// TwinCAT 3 PLC project Untitled1
// ProgramVersion: 3.1.4023.0
// libraries:
//   Tc2_Math, * (Beckhoff Automation GmbH)
//   Tc2_Standard, * (Beckhoff Automation GmbH)
//   Tc2_System, * (Beckhoff Automation GmbH)
//   Tc3_Mc3PlanarMotion, * (Beckhoff Automation GmbH)
//   Tc3_Module, * (Beckhoff Automation GmbH)
//   Tc3_Physics, * (Beckhoff Automation GmbH)
//   XboxControllerUtilities, * (Beckhoff Community)
// project tree:
//   / PlcTask.TcTTO
//   POUs/ MAIN.TcPOU
// real-time tasks:
//   TASK XPlanar Task3: cycle T#250us, priority 1, ADS port 350
//   TASK XPlanar Task4: cycle T#250us, priority 2, ADS port 351
//   TASK Job Task: cycle default, priority 32
//   TASK MC-Task (MET): cycle T#250us, priority 6, ADS port 521
//   TASK MC-Task (MPT): cycle T#10ms, priority 8, ADS port 531
//   TASK PlcTask: cycle T#250us, priority 20, ADS port 352
// I/O:
//   DEVICE Device 1 (EtherCAT) (disabled), AmsNetId 169.254.25.219.2.1
//     Term 1 (EK1200) [EK1200-5000 EtherCAT Power supply (2A E-Bus)]
//       Term 2 (EL9222-9482) [EL9222-9482 Overcurrent protection 24V DC, 2Ch., 8A/2A]
//       Term 3 (EL9222-6600) [EL9222-6600 Overcurrent protection 24V DC, 2Ch., max. 4A, adjustable]
//       Term 4 (EL9011) [EL9011 End Terminal]
//   DEVICE Device 6 (EtherCAT), AmsNetId 169.254.25.219.7.1
//     Term 5 (APS4322-7000) [APS4322-7000 Drive]
//       Term 6 (APS4322-5000) [APS4322-5000 Feedback]
//     Term 7 (APS4322-7000) [APS4322-7000 Drive]
//       Term 8 (APS4322-5000) [APS4322-5000 Feedback]
//     Term 9 (APS4322-7000) [APS4322-7000 Drive]
//       Term 10 (APS4322-5000) [APS4322-5000 Feedback]
//     Term 11 (APS4322-7000) [APS4322-7000 Drive]
//       Term 12 (APS4322-5000) [APS4322-5000 Feedback]
//     Term 13 (APS4322-7000) [APS4322-7000 Drive]
//       Term 14 (APS4322-5000) [APS4322-5000 Feedback]
//     Term 15 (APS4322-7000) [APS4322-7000 Drive]
//       Term 16 (APS4322-5000) [APS4322-5000 Feedback]
//   DEVICE Device 2 (EtherCAT), AmsNetId 169.254.25.219.3.1
//     Term 17 (APS4322-7000) [APS4322-7000 Drive]
//       Term 18 (APS4322-5000) [APS4322-5000 Feedback]
//     Term 19 (APS4322-7000) [APS4322-7000 Drive]
//       Term 20 (APS4322-5000) [APS4322-5000 Feedback]
//     Term 21 (APS4322-7000) [APS4322-7000 Drive]
//       Term 22 (APS4322-5000) [APS4322-5000 Feedback]
//     Term 23 (APS4322-7000) [APS4322-7000 Drive]
//       Term 24 (APS4322-5000) [APS4322-5000 Feedback]
//     Term 25 (APS4322-7000) [APS4322-7000 Drive]
//       Term 26 (APS4322-5000) [APS4322-5000 Feedback]
//     Term 27 (APS4322-7000) [APS4322-7000 Drive]
//       Term 28 (APS4322-5000) [APS4322-5000 Feedback]
// variable links:
//   Device 2 (EtherCAT) <-> TcCOM Objects/XPlanar/Part1/Tile1
//     Term 17 (APS4322-7000)/APS Comm Inputs/CommStatusWord <-> Data Pointer/MoverCommStatusWord
//     Term 17 (APS4322-7000)/APS Comm Inputs/Data {1..4} <-> Data Pointer/MoverCommDataIn[{0..3}]  (4 links)
//     Term 17 (APS4322-7000)/APS Comm Outputs/CommControlWord <-> Data Pointer/MoverCommControlWord
//     Term 17 (APS4322-7000)/APS Comm Outputs/Data 1 <-> Data Pointer/MoverCommDataOut
//     Term 17 (APS4322-7000)/APS Diagdata/DC Link Voltage <-> Data Pointer/DcLinkVoltage
//     Term 17 (APS4322-7000)/APS Diagdata/Power supply current <-> Data Pointer/PowerSupplyCurrent
//     Term 17 (APS4322-7000)/APS Inputs/StatusWord <-> Data Pointer/PowerUnitStatusWord
//     Term 17 (APS4322-7000)/APS Outputs/ControlWord <-> Data Pointer/PowerUnitControlWord
//     Term 17 (APS4322-7000)/APS Outputs/Current D 0X0 <-> Data Pointer/DCurrentSetPoints[0]
//     Term 17 (APS4322-7000)/APS Outputs/Current D 0X1 <-> Data Pointer/DCurrentSetPoints[1]
//     Term 17 (APS4322-7000)/APS Outputs/Current D 0X2 <-> Data Pointer/DCurrentSetPoints[2]
//     Term 17 (APS4322-7000)/APS Outputs/Current D 1X0 <-> Data Pointer/DCurrentSetPoints[6]
//     Term 17 (APS4322-7000)/APS Outputs/Current D 1X1 <-> Data Pointer/DCurrentSetPoints[7]
//     Term 17 (APS4322-7000)/APS Outputs/Current D 1X2 <-> Data Pointer/DCurrentSetPoints[8]
//     Term 17 (APS4322-7000)/APS Outputs/Current D 2X0 <-> Data Pointer/DCurrentSetPoints[12]
//     Term 17 (APS4322-7000)/APS Outputs/Current D 2X1 <-> Data Pointer/DCurrentSetPoints[13]
//     Term 17 (APS4322-7000)/APS Outputs/Current D 2X2 <-> Data Pointer/DCurrentSetPoints[14]
//     Term 17 (APS4322-7000)/APS Outputs/Current D 3X0 <-> Data Pointer/DCurrentSetPoints[18]
//     Term 17 (APS4322-7000)/APS Outputs/Current D 3X1 <-> Data Pointer/DCurrentSetPoints[19]
//     Term 17 (APS4322-7000)/APS Outputs/Current D 3X2 <-> Data Pointer/DCurrentSetPoints[20]
//     Term 17 (APS4322-7000)/APS Outputs/Current D 0Y0 <-> Data Pointer/DCurrentSetPoints[3]
//     Term 17 (APS4322-7000)/APS Outputs/Current D 0Y1 <-> Data Pointer/DCurrentSetPoints[4]
//     Term 17 (APS4322-7000)/APS Outputs/Current D 0Y2 <-> Data Pointer/DCurrentSetPoints[5]
//     Term 17 (APS4322-7000)/APS Outputs/Current D 1Y0 <-> Data Pointer/DCurrentSetPoints[9]
//     Term 17 (APS4322-7000)/APS Outputs/Current D 1Y1 <-> Data Pointer/DCurrentSetPoints[10]
//     Term 17 (APS4322-7000)/APS Outputs/Current D 1Y2 <-> Data Pointer/DCurrentSetPoints[11]
//     Term 17 (APS4322-7000)/APS Outputs/Current D 2Y0 <-> Data Pointer/DCurrentSetPoints[15]
//     Term 17 (APS4322-7000)/APS Outputs/Current D 2Y1 <-> Data Pointer/DCurrentSetPoints[16]
//     Term 17 (APS4322-7000)/APS Outputs/Current D 2Y2 <-> Data Pointer/DCurrentSetPoints[17]
//     Term 17 (APS4322-7000)/APS Outputs/Current D 3Y0 <-> Data Pointer/DCurrentSetPoints[21]
//     Term 17 (APS4322-7000)/APS Outputs/Current D 3Y1 <-> Data Pointer/DCurrentSetPoints[22]
//     Term 17 (APS4322-7000)/APS Outputs/Current D 3Y2 <-> Data Pointer/DCurrentSetPoints[23]
//     Term 17 (APS4322-7000)/APS Outputs/Current Q 0X0 <-> Data Pointer/QCurrentSetPoints[0]
//     Term 17 (APS4322-7000)/APS Outputs/Current Q 0X1 <-> Data Pointer/QCurrentSetPoints[1]
//     Term 17 (APS4322-7000)/APS Outputs/Current Q 0X2 <-> Data Pointer/QCurrentSetPoints[2]
//     Term 17 (APS4322-7000)/APS Outputs/Current Q 1X0 <-> Data Pointer/QCurrentSetPoints[6]
//     Term 17 (APS4322-7000)/APS Outputs/Current Q 1X1 <-> Data Pointer/QCurrentSetPoints[7]
//     Term 17 (APS4322-7000)/APS Outputs/Current Q 1X2 <-> Data Pointer/QCurrentSetPoints[8]
//     Term 17 (APS4322-7000)/APS Outputs/Current Q 2X0 <-> Data Pointer/QCurrentSetPoints[12]
//     Term 17 (APS4322-7000)/APS Outputs/Current Q 2X1 <-> Data Pointer/QCurrentSetPoints[13]
//     Term 17 (APS4322-7000)/APS Outputs/Current Q 2X2 <-> Data Pointer/QCurrentSetPoints[14]
//     Term 17 (APS4322-7000)/APS Outputs/Current Q 3X0 <-> Data Pointer/QCurrentSetPoints[18]
//     Term 17 (APS4322-7000)/APS Outputs/Current Q 3X1 <-> Data Pointer/QCurrentSetPoints[19]
//     Term 17 (APS4322-7000)/APS Outputs/Current Q 3X2 <-> Data Pointer/QCurrentSetPoints[20]
//     Term 17 (APS4322-7000)/APS Outputs/Current Q 0Y0 <-> Data Pointer/QCurrentSetPoints[3]
//     Term 17 (APS4322-7000)/APS Outputs/Current Q 0Y1 <-> Data Pointer/QCurrentSetPoints[4]
//     Term 17 (APS4322-7000)/APS Outputs/Current Q 0Y2 <-> Data Pointer/QCurrentSetPoints[5]
//     Term 17 (APS4322-7000)/APS Outputs/Current Q 1Y0 <-> Data Pointer/QCurrentSetPoints[9]
//     Term 17 (APS4322-7000)/APS Outputs/Current Q 1Y1 <-> Data Pointer/QCurrentSetPoints[10]
//     Term 17 (APS4322-7000)/APS Outputs/Current Q 1Y2 <-> Data Pointer/QCurrentSetPoints[11]
//     Term 17 (APS4322-7000)/APS Outputs/Current Q 2Y0 <-> Data Pointer/QCurrentSetPoints[15]
//     Term 17 (APS4322-7000)/APS Outputs/Current Q 2Y1 <-> Data Pointer/QCurrentSetPoints[16]
//     Term 17 (APS4322-7000)/APS Outputs/Current Q 2Y2 <-> Data Pointer/QCurrentSetPoints[17]
//     Term 17 (APS4322-7000)/APS Outputs/Current Q 3Y0 <-> Data Pointer/QCurrentSetPoints[21]
//     Term 17 (APS4322-7000)/APS Outputs/Current Q 3Y1 <-> Data Pointer/QCurrentSetPoints[22]
//     Term 17 (APS4322-7000)/APS Outputs/Current Q 3Y2 <-> Data Pointer/QCurrentSetPoints[23]
//     Term 17 (APS4322-7000)/APS Outputs/PhiE 0X0 <-> Data Pointer/PhiSetPoints[0]
//     Term 17 (APS4322-7000)/APS Outputs/PhiE 0X1 <-> Data Pointer/PhiSetPoints[1]
//     Term 17 (APS4322-7000)/APS Outputs/PhiE 0X2 <-> Data Pointer/PhiSetPoints[2]
//     Term 17 (APS4322-7000)/APS Outputs/PhiE 1X0 <-> Data Pointer/PhiSetPoints[6]
//     Term 17 (APS4322-7000)/APS Outputs/PhiE 1X1 <-> Data Pointer/PhiSetPoints[7]
//     Term 17 (APS4322-7000)/APS Outputs/PhiE 1X2 <-> Data Pointer/PhiSetPoints[8]
//     Term 17 (APS4322-7000)/APS Outputs/PhiE 2X0 <-> Data Pointer/PhiSetPoints[12]
//     Term 17 (APS4322-7000)/APS Outputs/PhiE 2X1 <-> Data Pointer/PhiSetPoints[13]
//     Term 17 (APS4322-7000)/APS Outputs/PhiE 2X2 <-> Data Pointer/PhiSetPoints[14]
//     Term 17 (APS4322-7000)/APS Outputs/PhiE 3X0 <-> Data Pointer/PhiSetPoints[18]
//     Term 17 (APS4322-7000)/APS Outputs/PhiE 3X1 <-> Data Pointer/PhiSetPoints[19]
//     Term 17 (APS4322-7000)/APS Outputs/PhiE 3X2 <-> Data Pointer/PhiSetPoints[20]
//     Term 17 (APS4322-7000)/APS Outputs/PhiE 0Y0 <-> Data Pointer/PhiSetPoints[3]
//     Term 17 (APS4322-7000)/APS Outputs/PhiE 0Y1 <-> Data Pointer/PhiSetPoints[4]
//     Term 17 (APS4322-7000)/APS Outputs/PhiE 0Y2 <-> Data Pointer/PhiSetPoints[5]
//     Term 17 (APS4322-7000)/APS Outputs/PhiE 1Y0 <-> Data Pointer/PhiSetPoints[9]
//     Term 17 (APS4322-7000)/APS Outputs/PhiE 1Y1 <-> Data Pointer/PhiSetPoints[10]
//     Term 17 (APS4322-7000)/APS Outputs/PhiE 1Y2 <-> Data Pointer/PhiSetPoints[11]
//     Term 17 (APS4322-7000)/APS Outputs/PhiE 2Y0 <-> Data Pointer/PhiSetPoints[15]
//     Term 17 (APS4322-7000)/APS Outputs/PhiE 2Y1 <-> Data Pointer/PhiSetPoints[16]
//     Term 17 (APS4322-7000)/APS Outputs/PhiE 2Y2 <-> Data Pointer/PhiSetPoints[17]
//     Term 17 (APS4322-7000)/APS Outputs/PhiE 3Y0 <-> Data Pointer/PhiSetPoints[21]
//     Term 17 (APS4322-7000)/APS Outputs/PhiE 3Y1 <-> Data Pointer/PhiSetPoints[22]
//     Term 17 (APS4322-7000)/APS Outputs/PhiE 3Y2 <-> Data Pointer/PhiSetPoints[23]
//     Term 17 (APS4322-7000)/Term 18 (APS4322-5000)/FB Inputs/A{0..8 step 2} X-Field <-> Data Pointer/HallSensorFieldsXYZ[{0..12 step 3}]  (5 links)
//     Term 17 (APS4322-7000)/Term 18 (APS4322-5000)/FB Inputs/A{0..8 step 2} Y-Field <-> Data Pointer/HallSensorFieldsXYZ[{1..13 step 3}]  (5 links)
//     Term 17 (APS4322-7000)/Term 18 (APS4322-5000)/FB Inputs/A{0..8 step 2} Z-Field <-> Data Pointer/HallSensorFieldsXYZ[{2..14 step 3}]  (5 links)
//     Term 17 (APS4322-7000)/Term 18 (APS4322-5000)/FB Inputs/B{1..9 step 2} X-Field <-> Data Pointer/HallSensorFieldsXYZ[{15..27 step 3}]  (5 links)
//     Term 17 (APS4322-7000)/Term 18 (APS4322-5000)/FB Inputs/B{1..9 step 2} Y-Field <-> Data Pointer/HallSensorFieldsXYZ[{16..28 step 3}]  (5 links)
//     Term 17 (APS4322-7000)/Term 18 (APS4322-5000)/FB Inputs/B{1..9 step 2} Z-Field <-> Data Pointer/HallSensorFieldsXYZ[{17..29 step 3}]  (5 links)
//     Term 17 (APS4322-7000)/Term 18 (APS4322-5000)/FB Inputs/C{0..8 step 2} X-Field <-> Data Pointer/HallSensorFieldsXYZ[{30..42 step 3}]  (5 links)
//     Term 17 (APS4322-7000)/Term 18 (APS4322-5000)/FB Inputs/C{0..8 step 2} Y-Field <-> Data Pointer/HallSensorFieldsXYZ[{31..43 step 3}]  (5 links)
//     Term 17 (APS4322-7000)/Term 18 (APS4322-5000)/FB Inputs/C{0..8 step 2} Z-Field <-> Data Pointer/HallSensorFieldsXYZ[{32..44 step 3}]  (5 links)
//     Term 17 (APS4322-7000)/Term 18 (APS4322-5000)/FB Inputs/D{1..9 step 2} X-Field <-> Data Pointer/HallSensorFieldsXYZ[{45..57 step 3}]  (5 links)
//     Term 17 (APS4322-7000)/Term 18 (APS4322-5000)/FB Inputs/D{1..9 step 2} Y-Field <-> Data Pointer/HallSensorFieldsXYZ[{46..58 step 3}]  (5 links)
//     Term 17 (APS4322-7000)/Term 18 (APS4322-5000)/FB Inputs/D{1..9 step 2} Z-Field <-> Data Pointer/HallSensorFieldsXYZ[{47..59 step 3}]  (5 links)
//     Term 17 (APS4322-7000)/Term 18 (APS4322-5000)/FB Inputs/E{0..8 step 2} X-Field <-> Data Pointer/HallSensorFieldsXYZ[{60..72 step 3}]  (5 links)
//     Term 17 (APS4322-7000)/Term 18 (APS4322-5000)/FB Inputs/E{0..8 step 2} Y-Field <-> Data Pointer/HallSensorFieldsXYZ[{61..73 step 3}]  (5 links)
//     Term 17 (APS4322-7000)/Term 18 (APS4322-5000)/FB Inputs/E{0..8 step 2} Z-Field <-> Data Pointer/HallSensorFieldsXYZ[{62..74 step 3}]  (5 links)
//     Term 17 (APS4322-7000)/Term 18 (APS4322-5000)/FB Inputs/F{1..9 step 2} X-Field <-> Data Pointer/HallSensorFieldsXYZ[{75..87 step 3}]  (5 links)
//     Term 17 (APS4322-7000)/Term 18 (APS4322-5000)/FB Inputs/F{1..9 step 2} Y-Field <-> Data Pointer/HallSensorFieldsXYZ[{76..88 step 3}]  (5 links)
//     Term 17 (APS4322-7000)/Term 18 (APS4322-5000)/FB Inputs/F{1..9 step 2} Z-Field <-> Data Pointer/HallSensorFieldsXYZ[{77..89 step 3}]  (5 links)
//     Term 17 (APS4322-7000)/Term 18 (APS4322-5000)/FB Inputs/G{0..8 step 2} X-Field <-> Data Pointer/HallSensorFieldsXYZ[{90..102 step 3}]  (5 links)
//     Term 17 (APS4322-7000)/Term 18 (APS4322-5000)/FB Inputs/G{0..8 step 2} Y-Field <-> Data Pointer/HallSensorFieldsXYZ[{91..103 step 3}]  (5 links)
//     Term 17 (APS4322-7000)/Term 18 (APS4322-5000)/FB Inputs/G{0..8 step 2} Z-Field <-> Data Pointer/HallSensorFieldsXYZ[{92..104 step 3}]  (5 links)
//     Term 17 (APS4322-7000)/Term 18 (APS4322-5000)/FB Inputs/H{1..9 step 2} X-Field <-> Data Pointer/HallSensorFieldsXYZ[{105..117 step 3}]  (5 links)
//     Term 17 (APS4322-7000)/Term 18 (APS4322-5000)/FB Inputs/H{1..9 step 2} Y-Field <-> Data Pointer/HallSensorFieldsXYZ[{106..118 step 3}]  (5 links)
//     Term 17 (APS4322-7000)/Term 18 (APS4322-5000)/FB Inputs/H{1..9 step 2} Z-Field <-> Data Pointer/HallSensorFieldsXYZ[{107..119 step 3}]  (5 links)
//     Term 17 (APS4322-7000)/Term 18 (APS4322-5000)/FB Inputs/I{0..8 step 2} X-Field <-> Data Pointer/HallSensorFieldsXYZ[{120..132 step 3}]  (5 links)
//     Term 17 (APS4322-7000)/Term 18 (APS4322-5000)/FB Inputs/I{0..8 step 2} Y-Field <-> Data Pointer/HallSensorFieldsXYZ[{121..133 step 3}]  (5 links)
//     Term 17 (APS4322-7000)/Term 18 (APS4322-5000)/FB Inputs/I{0..8 step 2} Z-Field <-> Data Pointer/HallSensorFieldsXYZ[{122..134 step 3}]  (5 links)
//     Term 17 (APS4322-7000)/Term 18 (APS4322-5000)/FB Inputs/J{1..9 step 2} X-Field <-> Data Pointer/HallSensorFieldsXYZ[{135..147 step 3}]  (5 links)
//     Term 17 (APS4322-7000)/Term 18 (APS4322-5000)/FB Inputs/J{1..9 step 2} Y-Field <-> Data Pointer/HallSensorFieldsXYZ[{136..148 step 3}]  (5 links)
//     Term 17 (APS4322-7000)/Term 18 (APS4322-5000)/FB Inputs/J{1..9 step 2} Z-Field <-> Data Pointer/HallSensorFieldsXYZ[{137..149 step 3}]  (5 links)
//     Term 17 (APS4322-7000)/Term 18 (APS4322-5000)/FB Inputs/Status <-> Data Pointer/FeedbackStatus
//   Device 2 (EtherCAT) <-> TcCOM Objects/XPlanar/Part1/Tile10
//     Term 27 (APS4322-7000)/APS Comm Inputs/CommStatusWord <-> Data Pointer/MoverCommStatusWord
//     Term 27 (APS4322-7000)/APS Comm Inputs/Data {1..4} <-> Data Pointer/MoverCommDataIn[{0..3}]  (4 links)
//     Term 27 (APS4322-7000)/APS Comm Outputs/CommControlWord <-> Data Pointer/MoverCommControlWord
//     Term 27 (APS4322-7000)/APS Comm Outputs/Data 1 <-> Data Pointer/MoverCommDataOut
//     Term 27 (APS4322-7000)/APS Diagdata/DC Link Voltage <-> Data Pointer/DcLinkVoltage
//     Term 27 (APS4322-7000)/APS Diagdata/Power supply current <-> Data Pointer/PowerSupplyCurrent
//     Term 27 (APS4322-7000)/APS Inputs/StatusWord <-> Data Pointer/PowerUnitStatusWord
//     Term 27 (APS4322-7000)/APS Outputs/ControlWord <-> Data Pointer/PowerUnitControlWord
//     Term 27 (APS4322-7000)/APS Outputs/Current D 0X0 <-> Data Pointer/DCurrentSetPoints[0]
//     Term 27 (APS4322-7000)/APS Outputs/Current D 0X1 <-> Data Pointer/DCurrentSetPoints[1]
//     Term 27 (APS4322-7000)/APS Outputs/Current D 0X2 <-> Data Pointer/DCurrentSetPoints[2]
//     Term 27 (APS4322-7000)/APS Outputs/Current D 1X0 <-> Data Pointer/DCurrentSetPoints[6]
//     Term 27 (APS4322-7000)/APS Outputs/Current D 1X1 <-> Data Pointer/DCurrentSetPoints[7]
//     Term 27 (APS4322-7000)/APS Outputs/Current D 1X2 <-> Data Pointer/DCurrentSetPoints[8]
//     Term 27 (APS4322-7000)/APS Outputs/Current D 2X0 <-> Data Pointer/DCurrentSetPoints[12]
//     Term 27 (APS4322-7000)/APS Outputs/Current D 2X1 <-> Data Pointer/DCurrentSetPoints[13]
//     Term 27 (APS4322-7000)/APS Outputs/Current D 2X2 <-> Data Pointer/DCurrentSetPoints[14]
//     Term 27 (APS4322-7000)/APS Outputs/Current D 3X0 <-> Data Pointer/DCurrentSetPoints[18]
//     Term 27 (APS4322-7000)/APS Outputs/Current D 3X1 <-> Data Pointer/DCurrentSetPoints[19]
//     Term 27 (APS4322-7000)/APS Outputs/Current D 3X2 <-> Data Pointer/DCurrentSetPoints[20]
//     Term 27 (APS4322-7000)/APS Outputs/Current D 0Y0 <-> Data Pointer/DCurrentSetPoints[3]
//     Term 27 (APS4322-7000)/APS Outputs/Current D 0Y1 <-> Data Pointer/DCurrentSetPoints[4]
//     Term 27 (APS4322-7000)/APS Outputs/Current D 0Y2 <-> Data Pointer/DCurrentSetPoints[5]
//     Term 27 (APS4322-7000)/APS Outputs/Current D 1Y0 <-> Data Pointer/DCurrentSetPoints[9]
//     Term 27 (APS4322-7000)/APS Outputs/Current D 1Y1 <-> Data Pointer/DCurrentSetPoints[10]
//     Term 27 (APS4322-7000)/APS Outputs/Current D 1Y2 <-> Data Pointer/DCurrentSetPoints[11]
//     Term 27 (APS4322-7000)/APS Outputs/Current D 2Y0 <-> Data Pointer/DCurrentSetPoints[15]
//     Term 27 (APS4322-7000)/APS Outputs/Current D 2Y1 <-> Data Pointer/DCurrentSetPoints[16]
//     Term 27 (APS4322-7000)/APS Outputs/Current D 2Y2 <-> Data Pointer/DCurrentSetPoints[17]
//     Term 27 (APS4322-7000)/APS Outputs/Current D 3Y0 <-> Data Pointer/DCurrentSetPoints[21]
//     Term 27 (APS4322-7000)/APS Outputs/Current D 3Y1 <-> Data Pointer/DCurrentSetPoints[22]
//     Term 27 (APS4322-7000)/APS Outputs/Current D 3Y2 <-> Data Pointer/DCurrentSetPoints[23]
//     Term 27 (APS4322-7000)/APS Outputs/Current Q 0X0 <-> Data Pointer/QCurrentSetPoints[0]
//     Term 27 (APS4322-7000)/APS Outputs/Current Q 0X1 <-> Data Pointer/QCurrentSetPoints[1]
//     Term 27 (APS4322-7000)/APS Outputs/Current Q 0X2 <-> Data Pointer/QCurrentSetPoints[2]
//     Term 27 (APS4322-7000)/APS Outputs/Current Q 1X0 <-> Data Pointer/QCurrentSetPoints[6]
//     Term 27 (APS4322-7000)/APS Outputs/Current Q 1X1 <-> Data Pointer/QCurrentSetPoints[7]
//     Term 27 (APS4322-7000)/APS Outputs/Current Q 1X2 <-> Data Pointer/QCurrentSetPoints[8]
//     Term 27 (APS4322-7000)/APS Outputs/Current Q 2X0 <-> Data Pointer/QCurrentSetPoints[12]
//     Term 27 (APS4322-7000)/APS Outputs/Current Q 2X1 <-> Data Pointer/QCurrentSetPoints[13]
//     Term 27 (APS4322-7000)/APS Outputs/Current Q 2X2 <-> Data Pointer/QCurrentSetPoints[14]
//     Term 27 (APS4322-7000)/APS Outputs/Current Q 3X0 <-> Data Pointer/QCurrentSetPoints[18]
//     Term 27 (APS4322-7000)/APS Outputs/Current Q 3X1 <-> Data Pointer/QCurrentSetPoints[19]
//     Term 27 (APS4322-7000)/APS Outputs/Current Q 3X2 <-> Data Pointer/QCurrentSetPoints[20]
//     Term 27 (APS4322-7000)/APS Outputs/Current Q 0Y0 <-> Data Pointer/QCurrentSetPoints[3]
//     Term 27 (APS4322-7000)/APS Outputs/Current Q 0Y1 <-> Data Pointer/QCurrentSetPoints[4]
//     Term 27 (APS4322-7000)/APS Outputs/Current Q 0Y2 <-> Data Pointer/QCurrentSetPoints[5]
//     Term 27 (APS4322-7000)/APS Outputs/Current Q 1Y0 <-> Data Pointer/QCurrentSetPoints[9]
//     Term 27 (APS4322-7000)/APS Outputs/Current Q 1Y1 <-> Data Pointer/QCurrentSetPoints[10]
//     Term 27 (APS4322-7000)/APS Outputs/Current Q 1Y2 <-> Data Pointer/QCurrentSetPoints[11]
//     Term 27 (APS4322-7000)/APS Outputs/Current Q 2Y0 <-> Data Pointer/QCurrentSetPoints[15]
//     Term 27 (APS4322-7000)/APS Outputs/Current Q 2Y1 <-> Data Pointer/QCurrentSetPoints[16]
//     Term 27 (APS4322-7000)/APS Outputs/Current Q 2Y2 <-> Data Pointer/QCurrentSetPoints[17]
//     Term 27 (APS4322-7000)/APS Outputs/Current Q 3Y0 <-> Data Pointer/QCurrentSetPoints[21]
//     Term 27 (APS4322-7000)/APS Outputs/Current Q 3Y1 <-> Data Pointer/QCurrentSetPoints[22]
//     Term 27 (APS4322-7000)/APS Outputs/Current Q 3Y2 <-> Data Pointer/QCurrentSetPoints[23]
//     Term 27 (APS4322-7000)/APS Outputs/PhiE 0X0 <-> Data Pointer/PhiSetPoints[0]
//     Term 27 (APS4322-7000)/APS Outputs/PhiE 0X1 <-> Data Pointer/PhiSetPoints[1]
//     Term 27 (APS4322-7000)/APS Outputs/PhiE 0X2 <-> Data Pointer/PhiSetPoints[2]
//     Term 27 (APS4322-7000)/APS Outputs/PhiE 1X0 <-> Data Pointer/PhiSetPoints[6]
//     Term 27 (APS4322-7000)/APS Outputs/PhiE 1X1 <-> Data Pointer/PhiSetPoints[7]
//     Term 27 (APS4322-7000)/APS Outputs/PhiE 1X2 <-> Data Pointer/PhiSetPoints[8]
//     Term 27 (APS4322-7000)/APS Outputs/PhiE 2X0 <-> Data Pointer/PhiSetPoints[12]
//     Term 27 (APS4322-7000)/APS Outputs/PhiE 2X1 <-> Data Pointer/PhiSetPoints[13]
//     Term 27 (APS4322-7000)/APS Outputs/PhiE 2X2 <-> Data Pointer/PhiSetPoints[14]
//     Term 27 (APS4322-7000)/APS Outputs/PhiE 3X0 <-> Data Pointer/PhiSetPoints[18]
//     Term 27 (APS4322-7000)/APS Outputs/PhiE 3X1 <-> Data Pointer/PhiSetPoints[19]
//     Term 27 (APS4322-7000)/APS Outputs/PhiE 3X2 <-> Data Pointer/PhiSetPoints[20]
//     Term 27 (APS4322-7000)/APS Outputs/PhiE 0Y0 <-> Data Pointer/PhiSetPoints[3]
//     Term 27 (APS4322-7000)/APS Outputs/PhiE 0Y1 <-> Data Pointer/PhiSetPoints[4]
//     Term 27 (APS4322-7000)/APS Outputs/PhiE 0Y2 <-> Data Pointer/PhiSetPoints[5]
//     Term 27 (APS4322-7000)/APS Outputs/PhiE 1Y0 <-> Data Pointer/PhiSetPoints[9]
//     Term 27 (APS4322-7000)/APS Outputs/PhiE 1Y1 <-> Data Pointer/PhiSetPoints[10]
//     Term 27 (APS4322-7000)/APS Outputs/PhiE 1Y2 <-> Data Pointer/PhiSetPoints[11]
//     Term 27 (APS4322-7000)/APS Outputs/PhiE 2Y0 <-> Data Pointer/PhiSetPoints[15]
//     Term 27 (APS4322-7000)/APS Outputs/PhiE 2Y1 <-> Data Pointer/PhiSetPoints[16]
//     Term 27 (APS4322-7000)/APS Outputs/PhiE 2Y2 <-> Data Pointer/PhiSetPoints[17]
//     Term 27 (APS4322-7000)/APS Outputs/PhiE 3Y0 <-> Data Pointer/PhiSetPoints[21]
//     Term 27 (APS4322-7000)/APS Outputs/PhiE 3Y1 <-> Data Pointer/PhiSetPoints[22]
//     Term 27 (APS4322-7000)/APS Outputs/PhiE 3Y2 <-> Data Pointer/PhiSetPoints[23]
//     Term 27 (APS4322-7000)/Term 28 (APS4322-5000)/FB Inputs/A{0..8 step 2} X-Field <-> Data Pointer/HallSensorFieldsXYZ[{0..12 step 3}]  (5 links)
//     Term 27 (APS4322-7000)/Term 28 (APS4322-5000)/FB Inputs/A{0..8 step 2} Y-Field <-> Data Pointer/HallSensorFieldsXYZ[{1..13 step 3}]  (5 links)
//     Term 27 (APS4322-7000)/Term 28 (APS4322-5000)/FB Inputs/A{0..8 step 2} Z-Field <-> Data Pointer/HallSensorFieldsXYZ[{2..14 step 3}]  (5 links)
//     Term 27 (APS4322-7000)/Term 28 (APS4322-5000)/FB Inputs/B{1..9 step 2} X-Field <-> Data Pointer/HallSensorFieldsXYZ[{15..27 step 3}]  (5 links)
//     Term 27 (APS4322-7000)/Term 28 (APS4322-5000)/FB Inputs/B{1..9 step 2} Y-Field <-> Data Pointer/HallSensorFieldsXYZ[{16..28 step 3}]  (5 links)
//     Term 27 (APS4322-7000)/Term 28 (APS4322-5000)/FB Inputs/B{1..9 step 2} Z-Field <-> Data Pointer/HallSensorFieldsXYZ[{17..29 step 3}]  (5 links)
//     Term 27 (APS4322-7000)/Term 28 (APS4322-5000)/FB Inputs/C{0..8 step 2} X-Field <-> Data Pointer/HallSensorFieldsXYZ[{30..42 step 3}]  (5 links)
//     Term 27 (APS4322-7000)/Term 28 (APS4322-5000)/FB Inputs/C{0..8 step 2} Y-Field <-> Data Pointer/HallSensorFieldsXYZ[{31..43 step 3}]  (5 links)
//     Term 27 (APS4322-7000)/Term 28 (APS4322-5000)/FB Inputs/C{0..8 step 2} Z-Field <-> Data Pointer/HallSensorFieldsXYZ[{32..44 step 3}]  (5 links)
//     Term 27 (APS4322-7000)/Term 28 (APS4322-5000)/FB Inputs/D{1..9 step 2} X-Field <-> Data Pointer/HallSensorFieldsXYZ[{45..57 step 3}]  (5 links)
//     Term 27 (APS4322-7000)/Term 28 (APS4322-5000)/FB Inputs/D{1..9 step 2} Y-Field <-> Data Pointer/HallSensorFieldsXYZ[{46..58 step 3}]  (5 links)
//     Term 27 (APS4322-7000)/Term 28 (APS4322-5000)/FB Inputs/D{1..9 step 2} Z-Field <-> Data Pointer/HallSensorFieldsXYZ[{47..59 step 3}]  (5 links)
//     Term 27 (APS4322-7000)/Term 28 (APS4322-5000)/FB Inputs/E{0..8 step 2} X-Field <-> Data Pointer/HallSensorFieldsXYZ[{60..72 step 3}]  (5 links)
//     Term 27 (APS4322-7000)/Term 28 (APS4322-5000)/FB Inputs/E{0..8 step 2} Y-Field <-> Data Pointer/HallSensorFieldsXYZ[{61..73 step 3}]  (5 links)
//     Term 27 (APS4322-7000)/Term 28 (APS4322-5000)/FB Inputs/E{0..8 step 2} Z-Field <-> Data Pointer/HallSensorFieldsXYZ[{62..74 step 3}]  (5 links)
//     Term 27 (APS4322-7000)/Term 28 (APS4322-5000)/FB Inputs/F{1..9 step 2} X-Field <-> Data Pointer/HallSensorFieldsXYZ[{75..87 step 3}]  (5 links)
//     Term 27 (APS4322-7000)/Term 28 (APS4322-5000)/FB Inputs/F{1..9 step 2} Y-Field <-> Data Pointer/HallSensorFieldsXYZ[{76..88 step 3}]  (5 links)
//     Term 27 (APS4322-7000)/Term 28 (APS4322-5000)/FB Inputs/F{1..9 step 2} Z-Field <-> Data Pointer/HallSensorFieldsXYZ[{77..89 step 3}]  (5 links)
//     Term 27 (APS4322-7000)/Term 28 (APS4322-5000)/FB Inputs/G{0..8 step 2} X-Field <-> Data Pointer/HallSensorFieldsXYZ[{90..102 step 3}]  (5 links)
//     Term 27 (APS4322-7000)/Term 28 (APS4322-5000)/FB Inputs/G{0..8 step 2} Y-Field <-> Data Pointer/HallSensorFieldsXYZ[{91..103 step 3}]  (5 links)
//     Term 27 (APS4322-7000)/Term 28 (APS4322-5000)/FB Inputs/G{0..8 step 2} Z-Field <-> Data Pointer/HallSensorFieldsXYZ[{92..104 step 3}]  (5 links)
//     Term 27 (APS4322-7000)/Term 28 (APS4322-5000)/FB Inputs/H{1..9 step 2} X-Field <-> Data Pointer/HallSensorFieldsXYZ[{105..117 step 3}]  (5 links)
//     Term 27 (APS4322-7000)/Term 28 (APS4322-5000)/FB Inputs/H{1..9 step 2} Y-Field <-> Data Pointer/HallSensorFieldsXYZ[{106..118 step 3}]  (5 links)
//     Term 27 (APS4322-7000)/Term 28 (APS4322-5000)/FB Inputs/H{1..9 step 2} Z-Field <-> Data Pointer/HallSensorFieldsXYZ[{107..119 step 3}]  (5 links)
//     Term 27 (APS4322-7000)/Term 28 (APS4322-5000)/FB Inputs/I{0..8 step 2} X-Field <-> Data Pointer/HallSensorFieldsXYZ[{120..132 step 3}]  (5 links)
//     Term 27 (APS4322-7000)/Term 28 (APS4322-5000)/FB Inputs/I{0..8 step 2} Y-Field <-> Data Pointer/HallSensorFieldsXYZ[{121..133 step 3}]  (5 links)
//     Term 27 (APS4322-7000)/Term 28 (APS4322-5000)/FB Inputs/I{0..8 step 2} Z-Field <-> Data Pointer/HallSensorFieldsXYZ[{122..134 step 3}]  (5 links)
//     Term 27 (APS4322-7000)/Term 28 (APS4322-5000)/FB Inputs/J{1..9 step 2} X-Field <-> Data Pointer/HallSensorFieldsXYZ[{135..147 step 3}]  (5 links)
//     Term 27 (APS4322-7000)/Term 28 (APS4322-5000)/FB Inputs/J{1..9 step 2} Y-Field <-> Data Pointer/HallSensorFieldsXYZ[{136..148 step 3}]  (5 links)
//     Term 27 (APS4322-7000)/Term 28 (APS4322-5000)/FB Inputs/J{1..9 step 2} Z-Field <-> Data Pointer/HallSensorFieldsXYZ[{137..149 step 3}]  (5 links)
//     Term 27 (APS4322-7000)/Term 28 (APS4322-5000)/FB Inputs/Status <-> Data Pointer/FeedbackStatus
//   Device 2 (EtherCAT) <-> TcCOM Objects/XPlanar/Part1/Tile2
//     Term 19 (APS4322-7000)/APS Comm Inputs/CommStatusWord <-> Data Pointer/MoverCommStatusWord
//     Term 19 (APS4322-7000)/APS Comm Inputs/Data {1..4} <-> Data Pointer/MoverCommDataIn[{0..3}]  (4 links)
//     Term 19 (APS4322-7000)/APS Comm Outputs/CommControlWord <-> Data Pointer/MoverCommControlWord
//     Term 19 (APS4322-7000)/APS Comm Outputs/Data 1 <-> Data Pointer/MoverCommDataOut
//     Term 19 (APS4322-7000)/APS Diagdata/DC Link Voltage <-> Data Pointer/DcLinkVoltage
//     Term 19 (APS4322-7000)/APS Diagdata/Power supply current <-> Data Pointer/PowerSupplyCurrent
//     Term 19 (APS4322-7000)/APS Inputs/StatusWord <-> Data Pointer/PowerUnitStatusWord
//     Term 19 (APS4322-7000)/APS Outputs/ControlWord <-> Data Pointer/PowerUnitControlWord
//     Term 19 (APS4322-7000)/APS Outputs/Current D 0X0 <-> Data Pointer/DCurrentSetPoints[0]
//     Term 19 (APS4322-7000)/APS Outputs/Current D 0X1 <-> Data Pointer/DCurrentSetPoints[1]
//     Term 19 (APS4322-7000)/APS Outputs/Current D 0X2 <-> Data Pointer/DCurrentSetPoints[2]
//     Term 19 (APS4322-7000)/APS Outputs/Current D 1X0 <-> Data Pointer/DCurrentSetPoints[6]
//     Term 19 (APS4322-7000)/APS Outputs/Current D 1X1 <-> Data Pointer/DCurrentSetPoints[7]
//     Term 19 (APS4322-7000)/APS Outputs/Current D 1X2 <-> Data Pointer/DCurrentSetPoints[8]
//     Term 19 (APS4322-7000)/APS Outputs/Current D 2X0 <-> Data Pointer/DCurrentSetPoints[12]
//     Term 19 (APS4322-7000)/APS Outputs/Current D 2X1 <-> Data Pointer/DCurrentSetPoints[13]
//     Term 19 (APS4322-7000)/APS Outputs/Current D 2X2 <-> Data Pointer/DCurrentSetPoints[14]
//     Term 19 (APS4322-7000)/APS Outputs/Current D 3X0 <-> Data Pointer/DCurrentSetPoints[18]
//     Term 19 (APS4322-7000)/APS Outputs/Current D 3X1 <-> Data Pointer/DCurrentSetPoints[19]
//     Term 19 (APS4322-7000)/APS Outputs/Current D 3X2 <-> Data Pointer/DCurrentSetPoints[20]
//     Term 19 (APS4322-7000)/APS Outputs/Current D 0Y0 <-> Data Pointer/DCurrentSetPoints[3]
//     Term 19 (APS4322-7000)/APS Outputs/Current D 0Y1 <-> Data Pointer/DCurrentSetPoints[4]
//     Term 19 (APS4322-7000)/APS Outputs/Current D 0Y2 <-> Data Pointer/DCurrentSetPoints[5]
//     Term 19 (APS4322-7000)/APS Outputs/Current D 1Y0 <-> Data Pointer/DCurrentSetPoints[9]
//     Term 19 (APS4322-7000)/APS Outputs/Current D 1Y1 <-> Data Pointer/DCurrentSetPoints[10]
//     Term 19 (APS4322-7000)/APS Outputs/Current D 1Y2 <-> Data Pointer/DCurrentSetPoints[11]
//     Term 19 (APS4322-7000)/APS Outputs/Current D 2Y0 <-> Data Pointer/DCurrentSetPoints[15]
//     Term 19 (APS4322-7000)/APS Outputs/Current D 2Y1 <-> Data Pointer/DCurrentSetPoints[16]
//     Term 19 (APS4322-7000)/APS Outputs/Current D 2Y2 <-> Data Pointer/DCurrentSetPoints[17]
//     Term 19 (APS4322-7000)/APS Outputs/Current D 3Y0 <-> Data Pointer/DCurrentSetPoints[21]
//     Term 19 (APS4322-7000)/APS Outputs/Current D 3Y1 <-> Data Pointer/DCurrentSetPoints[22]
//     Term 19 (APS4322-7000)/APS Outputs/Current D 3Y2 <-> Data Pointer/DCurrentSetPoints[23]
//     Term 19 (APS4322-7000)/APS Outputs/Current Q 0X0 <-> Data Pointer/QCurrentSetPoints[0]
//     Term 19 (APS4322-7000)/APS Outputs/Current Q 0X1 <-> Data Pointer/QCurrentSetPoints[1]
//     Term 19 (APS4322-7000)/APS Outputs/Current Q 0X2 <-> Data Pointer/QCurrentSetPoints[2]
//     Term 19 (APS4322-7000)/APS Outputs/Current Q 1X0 <-> Data Pointer/QCurrentSetPoints[6]
//     Term 19 (APS4322-7000)/APS Outputs/Current Q 1X1 <-> Data Pointer/QCurrentSetPoints[7]
//     Term 19 (APS4322-7000)/APS Outputs/Current Q 1X2 <-> Data Pointer/QCurrentSetPoints[8]
//     Term 19 (APS4322-7000)/APS Outputs/Current Q 2X0 <-> Data Pointer/QCurrentSetPoints[12]
//     Term 19 (APS4322-7000)/APS Outputs/Current Q 2X1 <-> Data Pointer/QCurrentSetPoints[13]
//     Term 19 (APS4322-7000)/APS Outputs/Current Q 2X2 <-> Data Pointer/QCurrentSetPoints[14]
//     Term 19 (APS4322-7000)/APS Outputs/Current Q 3X0 <-> Data Pointer/QCurrentSetPoints[18]
//     Term 19 (APS4322-7000)/APS Outputs/Current Q 3X1 <-> Data Pointer/QCurrentSetPoints[19]
//     Term 19 (APS4322-7000)/APS Outputs/Current Q 3X2 <-> Data Pointer/QCurrentSetPoints[20]
//     Term 19 (APS4322-7000)/APS Outputs/Current Q 0Y0 <-> Data Pointer/QCurrentSetPoints[3]
//     Term 19 (APS4322-7000)/APS Outputs/Current Q 0Y1 <-> Data Pointer/QCurrentSetPoints[4]
//     Term 19 (APS4322-7000)/APS Outputs/Current Q 0Y2 <-> Data Pointer/QCurrentSetPoints[5]
//     Term 19 (APS4322-7000)/APS Outputs/Current Q 1Y0 <-> Data Pointer/QCurrentSetPoints[9]
//     Term 19 (APS4322-7000)/APS Outputs/Current Q 1Y1 <-> Data Pointer/QCurrentSetPoints[10]
//     Term 19 (APS4322-7000)/APS Outputs/Current Q 1Y2 <-> Data Pointer/QCurrentSetPoints[11]
//     Term 19 (APS4322-7000)/APS Outputs/Current Q 2Y0 <-> Data Pointer/QCurrentSetPoints[15]
//     Term 19 (APS4322-7000)/APS Outputs/Current Q 2Y1 <-> Data Pointer/QCurrentSetPoints[16]
//     Term 19 (APS4322-7000)/APS Outputs/Current Q 2Y2 <-> Data Pointer/QCurrentSetPoints[17]
//     Term 19 (APS4322-7000)/APS Outputs/Current Q 3Y0 <-> Data Pointer/QCurrentSetPoints[21]
//     Term 19 (APS4322-7000)/APS Outputs/Current Q 3Y1 <-> Data Pointer/QCurrentSetPoints[22]
//     Term 19 (APS4322-7000)/APS Outputs/Current Q 3Y2 <-> Data Pointer/QCurrentSetPoints[23]
//     Term 19 (APS4322-7000)/APS Outputs/PhiE 0X0 <-> Data Pointer/PhiSetPoints[0]
//     Term 19 (APS4322-7000)/APS Outputs/PhiE 0X1 <-> Data Pointer/PhiSetPoints[1]
//     Term 19 (APS4322-7000)/APS Outputs/PhiE 0X2 <-> Data Pointer/PhiSetPoints[2]
//     Term 19 (APS4322-7000)/APS Outputs/PhiE 1X0 <-> Data Pointer/PhiSetPoints[6]
//     Term 19 (APS4322-7000)/APS Outputs/PhiE 1X1 <-> Data Pointer/PhiSetPoints[7]
//     Term 19 (APS4322-7000)/APS Outputs/PhiE 1X2 <-> Data Pointer/PhiSetPoints[8]
//     Term 19 (APS4322-7000)/APS Outputs/PhiE 2X0 <-> Data Pointer/PhiSetPoints[12]
//     Term 19 (APS4322-7000)/APS Outputs/PhiE 2X1 <-> Data Pointer/PhiSetPoints[13]
//     Term 19 (APS4322-7000)/APS Outputs/PhiE 2X2 <-> Data Pointer/PhiSetPoints[14]
//     Term 19 (APS4322-7000)/APS Outputs/PhiE 3X0 <-> Data Pointer/PhiSetPoints[18]
//     Term 19 (APS4322-7000)/APS Outputs/PhiE 3X1 <-> Data Pointer/PhiSetPoints[19]
//     Term 19 (APS4322-7000)/APS Outputs/PhiE 3X2 <-> Data Pointer/PhiSetPoints[20]
//     Term 19 (APS4322-7000)/APS Outputs/PhiE 0Y0 <-> Data Pointer/PhiSetPoints[3]
//     Term 19 (APS4322-7000)/APS Outputs/PhiE 0Y1 <-> Data Pointer/PhiSetPoints[4]
//     Term 19 (APS4322-7000)/APS Outputs/PhiE 0Y2 <-> Data Pointer/PhiSetPoints[5]
//     Term 19 (APS4322-7000)/APS Outputs/PhiE 1Y0 <-> Data Pointer/PhiSetPoints[9]
//     Term 19 (APS4322-7000)/APS Outputs/PhiE 1Y1 <-> Data Pointer/PhiSetPoints[10]
//     Term 19 (APS4322-7000)/APS Outputs/PhiE 1Y2 <-> Data Pointer/PhiSetPoints[11]
//     Term 19 (APS4322-7000)/APS Outputs/PhiE 2Y0 <-> Data Pointer/PhiSetPoints[15]
//     Term 19 (APS4322-7000)/APS Outputs/PhiE 2Y1 <-> Data Pointer/PhiSetPoints[16]
//     Term 19 (APS4322-7000)/APS Outputs/PhiE 2Y2 <-> Data Pointer/PhiSetPoints[17]
//     Term 19 (APS4322-7000)/APS Outputs/PhiE 3Y0 <-> Data Pointer/PhiSetPoints[21]
//     Term 19 (APS4322-7000)/APS Outputs/PhiE 3Y1 <-> Data Pointer/PhiSetPoints[22]
//     Term 19 (APS4322-7000)/APS Outputs/PhiE 3Y2 <-> Data Pointer/PhiSetPoints[23]
//     Term 19 (APS4322-7000)/Term 20 (APS4322-5000)/FB Inputs/A{0..8 step 2} X-Field <-> Data Pointer/HallSensorFieldsXYZ[{0..12 step 3}]  (5 links)
//     Term 19 (APS4322-7000)/Term 20 (APS4322-5000)/FB Inputs/A{0..8 step 2} Y-Field <-> Data Pointer/HallSensorFieldsXYZ[{1..13 step 3}]  (5 links)
//     Term 19 (APS4322-7000)/Term 20 (APS4322-5000)/FB Inputs/A{0..8 step 2} Z-Field <-> Data Pointer/HallSensorFieldsXYZ[{2..14 step 3}]  (5 links)
//     Term 19 (APS4322-7000)/Term 20 (APS4322-5000)/FB Inputs/B{1..9 step 2} X-Field <-> Data Pointer/HallSensorFieldsXYZ[{15..27 step 3}]  (5 links)
//     Term 19 (APS4322-7000)/Term 20 (APS4322-5000)/FB Inputs/B{1..9 step 2} Y-Field <-> Data Pointer/HallSensorFieldsXYZ[{16..28 step 3}]  (5 links)
//     Term 19 (APS4322-7000)/Term 20 (APS4322-5000)/FB Inputs/B{1..9 step 2} Z-Field <-> Data Pointer/HallSensorFieldsXYZ[{17..29 step 3}]  (5 links)
//     Term 19 (APS4322-7000)/Term 20 (APS4322-5000)/FB Inputs/C{0..8 step 2} X-Field <-> Data Pointer/HallSensorFieldsXYZ[{30..42 step 3}]  (5 links)
//     Term 19 (APS4322-7000)/Term 20 (APS4322-5000)/FB Inputs/C{0..8 step 2} Y-Field <-> Data Pointer/HallSensorFieldsXYZ[{31..43 step 3}]  (5 links)
//     Term 19 (APS4322-7000)/Term 20 (APS4322-5000)/FB Inputs/C{0..8 step 2} Z-Field <-> Data Pointer/HallSensorFieldsXYZ[{32..44 step 3}]  (5 links)
//     Term 19 (APS4322-7000)/Term 20 (APS4322-5000)/FB Inputs/D{1..9 step 2} X-Field <-> Data Pointer/HallSensorFieldsXYZ[{45..57 step 3}]  (5 links)
//     Term 19 (APS4322-7000)/Term 20 (APS4322-5000)/FB Inputs/D{1..9 step 2} Y-Field <-> Data Pointer/HallSensorFieldsXYZ[{46..58 step 3}]  (5 links)
//     Term 19 (APS4322-7000)/Term 20 (APS4322-5000)/FB Inputs/D{1..9 step 2} Z-Field <-> Data Pointer/HallSensorFieldsXYZ[{47..59 step 3}]  (5 links)
//     Term 19 (APS4322-7000)/Term 20 (APS4322-5000)/FB Inputs/E{0..8 step 2} X-Field <-> Data Pointer/HallSensorFieldsXYZ[{60..72 step 3}]  (5 links)
//     Term 19 (APS4322-7000)/Term 20 (APS4322-5000)/FB Inputs/E{0..8 step 2} Y-Field <-> Data Pointer/HallSensorFieldsXYZ[{61..73 step 3}]  (5 links)
//     Term 19 (APS4322-7000)/Term 20 (APS4322-5000)/FB Inputs/E{0..8 step 2} Z-Field <-> Data Pointer/HallSensorFieldsXYZ[{62..74 step 3}]  (5 links)
//     Term 19 (APS4322-7000)/Term 20 (APS4322-5000)/FB Inputs/F{1..9 step 2} X-Field <-> Data Pointer/HallSensorFieldsXYZ[{75..87 step 3}]  (5 links)
//     Term 19 (APS4322-7000)/Term 20 (APS4322-5000)/FB Inputs/F{1..9 step 2} Y-Field <-> Data Pointer/HallSensorFieldsXYZ[{76..88 step 3}]  (5 links)
//     Term 19 (APS4322-7000)/Term 20 (APS4322-5000)/FB Inputs/F{1..9 step 2} Z-Field <-> Data Pointer/HallSensorFieldsXYZ[{77..89 step 3}]  (5 links)
//     Term 19 (APS4322-7000)/Term 20 (APS4322-5000)/FB Inputs/G{0..8 step 2} X-Field <-> Data Pointer/HallSensorFieldsXYZ[{90..102 step 3}]  (5 links)
//     Term 19 (APS4322-7000)/Term 20 (APS4322-5000)/FB Inputs/G{0..8 step 2} Y-Field <-> Data Pointer/HallSensorFieldsXYZ[{91..103 step 3}]  (5 links)
//     Term 19 (APS4322-7000)/Term 20 (APS4322-5000)/FB Inputs/G{0..8 step 2} Z-Field <-> Data Pointer/HallSensorFieldsXYZ[{92..104 step 3}]  (5 links)
//     Term 19 (APS4322-7000)/Term 20 (APS4322-5000)/FB Inputs/H{1..9 step 2} X-Field <-> Data Pointer/HallSensorFieldsXYZ[{105..117 step 3}]  (5 links)
//     Term 19 (APS4322-7000)/Term 20 (APS4322-5000)/FB Inputs/H{1..9 step 2} Y-Field <-> Data Pointer/HallSensorFieldsXYZ[{106..118 step 3}]  (5 links)
//     Term 19 (APS4322-7000)/Term 20 (APS4322-5000)/FB Inputs/H{1..9 step 2} Z-Field <-> Data Pointer/HallSensorFieldsXYZ[{107..119 step 3}]  (5 links)
//     Term 19 (APS4322-7000)/Term 20 (APS4322-5000)/FB Inputs/I{0..8 step 2} X-Field <-> Data Pointer/HallSensorFieldsXYZ[{120..132 step 3}]  (5 links)
//     Term 19 (APS4322-7000)/Term 20 (APS4322-5000)/FB Inputs/I{0..8 step 2} Y-Field <-> Data Pointer/HallSensorFieldsXYZ[{121..133 step 3}]  (5 links)
//     Term 19 (APS4322-7000)/Term 20 (APS4322-5000)/FB Inputs/I{0..8 step 2} Z-Field <-> Data Pointer/HallSensorFieldsXYZ[{122..134 step 3}]  (5 links)
//     Term 19 (APS4322-7000)/Term 20 (APS4322-5000)/FB Inputs/J{1..9 step 2} X-Field <-> Data Pointer/HallSensorFieldsXYZ[{135..147 step 3}]  (5 links)
//     Term 19 (APS4322-7000)/Term 20 (APS4322-5000)/FB Inputs/J{1..9 step 2} Y-Field <-> Data Pointer/HallSensorFieldsXYZ[{136..148 step 3}]  (5 links)
//     Term 19 (APS4322-7000)/Term 20 (APS4322-5000)/FB Inputs/J{1..9 step 2} Z-Field <-> Data Pointer/HallSensorFieldsXYZ[{137..149 step 3}]  (5 links)
//     Term 19 (APS4322-7000)/Term 20 (APS4322-5000)/FB Inputs/Status <-> Data Pointer/FeedbackStatus
//   Device 2 (EtherCAT) <-> TcCOM Objects/XPlanar/Part1/Tile5
//     Term 21 (APS4322-7000)/APS Comm Inputs/CommStatusWord <-> Data Pointer/MoverCommStatusWord
//     Term 21 (APS4322-7000)/APS Comm Inputs/Data {1..4} <-> Data Pointer/MoverCommDataIn[{0..3}]  (4 links)
//     Term 21 (APS4322-7000)/APS Comm Outputs/CommControlWord <-> Data Pointer/MoverCommControlWord
//     Term 21 (APS4322-7000)/APS Comm Outputs/Data 1 <-> Data Pointer/MoverCommDataOut
//     Term 21 (APS4322-7000)/APS Diagdata/DC Link Voltage <-> Data Pointer/DcLinkVoltage
//     Term 21 (APS4322-7000)/APS Diagdata/Power supply current <-> Data Pointer/PowerSupplyCurrent
//     Term 21 (APS4322-7000)/APS Inputs/StatusWord <-> Data Pointer/PowerUnitStatusWord
//     Term 21 (APS4322-7000)/APS Outputs/ControlWord <-> Data Pointer/PowerUnitControlWord
//     Term 21 (APS4322-7000)/APS Outputs/Current D 0X0 <-> Data Pointer/DCurrentSetPoints[0]
//     Term 21 (APS4322-7000)/APS Outputs/Current D 0X1 <-> Data Pointer/DCurrentSetPoints[1]
//     Term 21 (APS4322-7000)/APS Outputs/Current D 0X2 <-> Data Pointer/DCurrentSetPoints[2]
//     Term 21 (APS4322-7000)/APS Outputs/Current D 1X0 <-> Data Pointer/DCurrentSetPoints[6]
//     Term 21 (APS4322-7000)/APS Outputs/Current D 1X1 <-> Data Pointer/DCurrentSetPoints[7]
//     Term 21 (APS4322-7000)/APS Outputs/Current D 1X2 <-> Data Pointer/DCurrentSetPoints[8]
//     Term 21 (APS4322-7000)/APS Outputs/Current D 2X0 <-> Data Pointer/DCurrentSetPoints[12]
//     Term 21 (APS4322-7000)/APS Outputs/Current D 2X1 <-> Data Pointer/DCurrentSetPoints[13]
//     Term 21 (APS4322-7000)/APS Outputs/Current D 2X2 <-> Data Pointer/DCurrentSetPoints[14]
//     Term 21 (APS4322-7000)/APS Outputs/Current D 3X0 <-> Data Pointer/DCurrentSetPoints[18]
//     Term 21 (APS4322-7000)/APS Outputs/Current D 3X1 <-> Data Pointer/DCurrentSetPoints[19]
//     Term 21 (APS4322-7000)/APS Outputs/Current D 3X2 <-> Data Pointer/DCurrentSetPoints[20]
//     Term 21 (APS4322-7000)/APS Outputs/Current D 0Y0 <-> Data Pointer/DCurrentSetPoints[3]
//     Term 21 (APS4322-7000)/APS Outputs/Current D 0Y1 <-> Data Pointer/DCurrentSetPoints[4]
//     Term 21 (APS4322-7000)/APS Outputs/Current D 0Y2 <-> Data Pointer/DCurrentSetPoints[5]
//     Term 21 (APS4322-7000)/APS Outputs/Current D 1Y0 <-> Data Pointer/DCurrentSetPoints[9]
//     Term 21 (APS4322-7000)/APS Outputs/Current D 1Y1 <-> Data Pointer/DCurrentSetPoints[10]
//     Term 21 (APS4322-7000)/APS Outputs/Current D 1Y2 <-> Data Pointer/DCurrentSetPoints[11]
//     Term 21 (APS4322-7000)/APS Outputs/Current D 2Y0 <-> Data Pointer/DCurrentSetPoints[15]
//     Term 21 (APS4322-7000)/APS Outputs/Current D 2Y1 <-> Data Pointer/DCurrentSetPoints[16]
//     Term 21 (APS4322-7000)/APS Outputs/Current D 2Y2 <-> Data Pointer/DCurrentSetPoints[17]
//     Term 21 (APS4322-7000)/APS Outputs/Current D 3Y0 <-> Data Pointer/DCurrentSetPoints[21]
//     Term 21 (APS4322-7000)/APS Outputs/Current D 3Y1 <-> Data Pointer/DCurrentSetPoints[22]
//     Term 21 (APS4322-7000)/APS Outputs/Current D 3Y2 <-> Data Pointer/DCurrentSetPoints[23]
//     Term 21 (APS4322-7000)/APS Outputs/Current Q 0X0 <-> Data Pointer/QCurrentSetPoints[0]
//     Term 21 (APS4322-7000)/APS Outputs/Current Q 0X1 <-> Data Pointer/QCurrentSetPoints[1]
//     Term 21 (APS4322-7000)/APS Outputs/Current Q 0X2 <-> Data Pointer/QCurrentSetPoints[2]
//     Term 21 (APS4322-7000)/APS Outputs/Current Q 1X0 <-> Data Pointer/QCurrentSetPoints[6]
//     Term 21 (APS4322-7000)/APS Outputs/Current Q 1X1 <-> Data Pointer/QCurrentSetPoints[7]
//     Term 21 (APS4322-7000)/APS Outputs/Current Q 1X2 <-> Data Pointer/QCurrentSetPoints[8]
//     Term 21 (APS4322-7000)/APS Outputs/Current Q 2X0 <-> Data Pointer/QCurrentSetPoints[12]
//     Term 21 (APS4322-7000)/APS Outputs/Current Q 2X1 <-> Data Pointer/QCurrentSetPoints[13]
//     Term 21 (APS4322-7000)/APS Outputs/Current Q 2X2 <-> Data Pointer/QCurrentSetPoints[14]
//     Term 21 (APS4322-7000)/APS Outputs/Current Q 3X0 <-> Data Pointer/QCurrentSetPoints[18]
//     Term 21 (APS4322-7000)/APS Outputs/Current Q 3X1 <-> Data Pointer/QCurrentSetPoints[19]
//     Term 21 (APS4322-7000)/APS Outputs/Current Q 3X2 <-> Data Pointer/QCurrentSetPoints[20]
//     Term 21 (APS4322-7000)/APS Outputs/Current Q 0Y0 <-> Data Pointer/QCurrentSetPoints[3]
//     Term 21 (APS4322-7000)/APS Outputs/Current Q 0Y1 <-> Data Pointer/QCurrentSetPoints[4]
//     Term 21 (APS4322-7000)/APS Outputs/Current Q 0Y2 <-> Data Pointer/QCurrentSetPoints[5]
//     Term 21 (APS4322-7000)/APS Outputs/Current Q 1Y0 <-> Data Pointer/QCurrentSetPoints[9]
//     Term 21 (APS4322-7000)/APS Outputs/Current Q 1Y1 <-> Data Pointer/QCurrentSetPoints[10]
//     Term 21 (APS4322-7000)/APS Outputs/Current Q 1Y2 <-> Data Pointer/QCurrentSetPoints[11]
//     Term 21 (APS4322-7000)/APS Outputs/Current Q 2Y0 <-> Data Pointer/QCurrentSetPoints[15]
//     Term 21 (APS4322-7000)/APS Outputs/Current Q 2Y1 <-> Data Pointer/QCurrentSetPoints[16]
//     Term 21 (APS4322-7000)/APS Outputs/Current Q 2Y2 <-> Data Pointer/QCurrentSetPoints[17]
//     Term 21 (APS4322-7000)/APS Outputs/Current Q 3Y0 <-> Data Pointer/QCurrentSetPoints[21]
//     Term 21 (APS4322-7000)/APS Outputs/Current Q 3Y1 <-> Data Pointer/QCurrentSetPoints[22]
//     Term 21 (APS4322-7000)/APS Outputs/Current Q 3Y2 <-> Data Pointer/QCurrentSetPoints[23]
//     Term 21 (APS4322-7000)/APS Outputs/PhiE 0X0 <-> Data Pointer/PhiSetPoints[0]
//     Term 21 (APS4322-7000)/APS Outputs/PhiE 0X1 <-> Data Pointer/PhiSetPoints[1]
//     Term 21 (APS4322-7000)/APS Outputs/PhiE 0X2 <-> Data Pointer/PhiSetPoints[2]
//     Term 21 (APS4322-7000)/APS Outputs/PhiE 1X0 <-> Data Pointer/PhiSetPoints[6]
//     Term 21 (APS4322-7000)/APS Outputs/PhiE 1X1 <-> Data Pointer/PhiSetPoints[7]
//     Term 21 (APS4322-7000)/APS Outputs/PhiE 1X2 <-> Data Pointer/PhiSetPoints[8]
//     Term 21 (APS4322-7000)/APS Outputs/PhiE 2X0 <-> Data Pointer/PhiSetPoints[12]
//     Term 21 (APS4322-7000)/APS Outputs/PhiE 2X1 <-> Data Pointer/PhiSetPoints[13]
//     Term 21 (APS4322-7000)/APS Outputs/PhiE 2X2 <-> Data Pointer/PhiSetPoints[14]
//     Term 21 (APS4322-7000)/APS Outputs/PhiE 3X0 <-> Data Pointer/PhiSetPoints[18]
//     Term 21 (APS4322-7000)/APS Outputs/PhiE 3X1 <-> Data Pointer/PhiSetPoints[19]
//     Term 21 (APS4322-7000)/APS Outputs/PhiE 3X2 <-> Data Pointer/PhiSetPoints[20]
//     Term 21 (APS4322-7000)/APS Outputs/PhiE 0Y0 <-> Data Pointer/PhiSetPoints[3]
//     Term 21 (APS4322-7000)/APS Outputs/PhiE 0Y1 <-> Data Pointer/PhiSetPoints[4]
//     Term 21 (APS4322-7000)/APS Outputs/PhiE 0Y2 <-> Data Pointer/PhiSetPoints[5]
//     Term 21 (APS4322-7000)/APS Outputs/PhiE 1Y0 <-> Data Pointer/PhiSetPoints[9]
//     Term 21 (APS4322-7000)/APS Outputs/PhiE 1Y1 <-> Data Pointer/PhiSetPoints[10]
//     Term 21 (APS4322-7000)/APS Outputs/PhiE 1Y2 <-> Data Pointer/PhiSetPoints[11]
//     Term 21 (APS4322-7000)/APS Outputs/PhiE 2Y0 <-> Data Pointer/PhiSetPoints[15]
//     Term 21 (APS4322-7000)/APS Outputs/PhiE 2Y1 <-> Data Pointer/PhiSetPoints[16]
//     Term 21 (APS4322-7000)/APS Outputs/PhiE 2Y2 <-> Data Pointer/PhiSetPoints[17]
//     Term 21 (APS4322-7000)/APS Outputs/PhiE 3Y0 <-> Data Pointer/PhiSetPoints[21]
//     Term 21 (APS4322-7000)/APS Outputs/PhiE 3Y1 <-> Data Pointer/PhiSetPoints[22]
//     Term 21 (APS4322-7000)/APS Outputs/PhiE 3Y2 <-> Data Pointer/PhiSetPoints[23]
//     Term 21 (APS4322-7000)/Term 22 (APS4322-5000)/FB Inputs/A{0..8 step 2} X-Field <-> Data Pointer/HallSensorFieldsXYZ[{0..12 step 3}]  (5 links)
//     Term 21 (APS4322-7000)/Term 22 (APS4322-5000)/FB Inputs/A{0..8 step 2} Y-Field <-> Data Pointer/HallSensorFieldsXYZ[{1..13 step 3}]  (5 links)
//     Term 21 (APS4322-7000)/Term 22 (APS4322-5000)/FB Inputs/A{0..8 step 2} Z-Field <-> Data Pointer/HallSensorFieldsXYZ[{2..14 step 3}]  (5 links)
//     Term 21 (APS4322-7000)/Term 22 (APS4322-5000)/FB Inputs/B{1..9 step 2} X-Field <-> Data Pointer/HallSensorFieldsXYZ[{15..27 step 3}]  (5 links)
//     Term 21 (APS4322-7000)/Term 22 (APS4322-5000)/FB Inputs/B{1..9 step 2} Y-Field <-> Data Pointer/HallSensorFieldsXYZ[{16..28 step 3}]  (5 links)
//     Term 21 (APS4322-7000)/Term 22 (APS4322-5000)/FB Inputs/B{1..9 step 2} Z-Field <-> Data Pointer/HallSensorFieldsXYZ[{17..29 step 3}]  (5 links)
//     Term 21 (APS4322-7000)/Term 22 (APS4322-5000)/FB Inputs/C{0..8 step 2} X-Field <-> Data Pointer/HallSensorFieldsXYZ[{30..42 step 3}]  (5 links)
//     Term 21 (APS4322-7000)/Term 22 (APS4322-5000)/FB Inputs/C{0..8 step 2} Y-Field <-> Data Pointer/HallSensorFieldsXYZ[{31..43 step 3}]  (5 links)
//     Term 21 (APS4322-7000)/Term 22 (APS4322-5000)/FB Inputs/C{0..8 step 2} Z-Field <-> Data Pointer/HallSensorFieldsXYZ[{32..44 step 3}]  (5 links)
//     Term 21 (APS4322-7000)/Term 22 (APS4322-5000)/FB Inputs/D{1..9 step 2} X-Field <-> Data Pointer/HallSensorFieldsXYZ[{45..57 step 3}]  (5 links)
//     Term 21 (APS4322-7000)/Term 22 (APS4322-5000)/FB Inputs/D{1..9 step 2} Y-Field <-> Data Pointer/HallSensorFieldsXYZ[{46..58 step 3}]  (5 links)
//     Term 21 (APS4322-7000)/Term 22 (APS4322-5000)/FB Inputs/D{1..9 step 2} Z-Field <-> Data Pointer/HallSensorFieldsXYZ[{47..59 step 3}]  (5 links)
//     Term 21 (APS4322-7000)/Term 22 (APS4322-5000)/FB Inputs/E{0..8 step 2} X-Field <-> Data Pointer/HallSensorFieldsXYZ[{60..72 step 3}]  (5 links)
//     Term 21 (APS4322-7000)/Term 22 (APS4322-5000)/FB Inputs/E{0..8 step 2} Y-Field <-> Data Pointer/HallSensorFieldsXYZ[{61..73 step 3}]  (5 links)
//     Term 21 (APS4322-7000)/Term 22 (APS4322-5000)/FB Inputs/E{0..8 step 2} Z-Field <-> Data Pointer/HallSensorFieldsXYZ[{62..74 step 3}]  (5 links)
//     Term 21 (APS4322-7000)/Term 22 (APS4322-5000)/FB Inputs/F{1..9 step 2} X-Field <-> Data Pointer/HallSensorFieldsXYZ[{75..87 step 3}]  (5 links)
//     Term 21 (APS4322-7000)/Term 22 (APS4322-5000)/FB Inputs/F{1..9 step 2} Y-Field <-> Data Pointer/HallSensorFieldsXYZ[{76..88 step 3}]  (5 links)
//     Term 21 (APS4322-7000)/Term 22 (APS4322-5000)/FB Inputs/F{1..9 step 2} Z-Field <-> Data Pointer/HallSensorFieldsXYZ[{77..89 step 3}]  (5 links)
//     Term 21 (APS4322-7000)/Term 22 (APS4322-5000)/FB Inputs/G{0..8 step 2} X-Field <-> Data Pointer/HallSensorFieldsXYZ[{90..102 step 3}]  (5 links)
//     Term 21 (APS4322-7000)/Term 22 (APS4322-5000)/FB Inputs/G{0..8 step 2} Y-Field <-> Data Pointer/HallSensorFieldsXYZ[{91..103 step 3}]  (5 links)
//     Term 21 (APS4322-7000)/Term 22 (APS4322-5000)/FB Inputs/G{0..8 step 2} Z-Field <-> Data Pointer/HallSensorFieldsXYZ[{92..104 step 3}]  (5 links)
//     Term 21 (APS4322-7000)/Term 22 (APS4322-5000)/FB Inputs/H{1..9 step 2} X-Field <-> Data Pointer/HallSensorFieldsXYZ[{105..117 step 3}]  (5 links)
//     Term 21 (APS4322-7000)/Term 22 (APS4322-5000)/FB Inputs/H{1..9 step 2} Y-Field <-> Data Pointer/HallSensorFieldsXYZ[{106..118 step 3}]  (5 links)
//     Term 21 (APS4322-7000)/Term 22 (APS4322-5000)/FB Inputs/H{1..9 step 2} Z-Field <-> Data Pointer/HallSensorFieldsXYZ[{107..119 step 3}]  (5 links)
//     Term 21 (APS4322-7000)/Term 22 (APS4322-5000)/FB Inputs/I{0..8 step 2} X-Field <-> Data Pointer/HallSensorFieldsXYZ[{120..132 step 3}]  (5 links)
//     Term 21 (APS4322-7000)/Term 22 (APS4322-5000)/FB Inputs/I{0..8 step 2} Y-Field <-> Data Pointer/HallSensorFieldsXYZ[{121..133 step 3}]  (5 links)
//     Term 21 (APS4322-7000)/Term 22 (APS4322-5000)/FB Inputs/I{0..8 step 2} Z-Field <-> Data Pointer/HallSensorFieldsXYZ[{122..134 step 3}]  (5 links)
//     Term 21 (APS4322-7000)/Term 22 (APS4322-5000)/FB Inputs/J{1..9 step 2} X-Field <-> Data Pointer/HallSensorFieldsXYZ[{135..147 step 3}]  (5 links)
//     Term 21 (APS4322-7000)/Term 22 (APS4322-5000)/FB Inputs/J{1..9 step 2} Y-Field <-> Data Pointer/HallSensorFieldsXYZ[{136..148 step 3}]  (5 links)
//     Term 21 (APS4322-7000)/Term 22 (APS4322-5000)/FB Inputs/J{1..9 step 2} Z-Field <-> Data Pointer/HallSensorFieldsXYZ[{137..149 step 3}]  (5 links)
//     Term 21 (APS4322-7000)/Term 22 (APS4322-5000)/FB Inputs/Status <-> Data Pointer/FeedbackStatus
//   Device 2 (EtherCAT) <-> TcCOM Objects/XPlanar/Part1/Tile6
//     Term 23 (APS4322-7000)/APS Comm Inputs/CommStatusWord <-> Data Pointer/MoverCommStatusWord
//     Term 23 (APS4322-7000)/APS Comm Inputs/Data {1..4} <-> Data Pointer/MoverCommDataIn[{0..3}]  (4 links)
//     Term 23 (APS4322-7000)/APS Comm Outputs/CommControlWord <-> Data Pointer/MoverCommControlWord
//     Term 23 (APS4322-7000)/APS Comm Outputs/Data 1 <-> Data Pointer/MoverCommDataOut
//     Term 23 (APS4322-7000)/APS Diagdata/DC Link Voltage <-> Data Pointer/DcLinkVoltage
//     Term 23 (APS4322-7000)/APS Diagdata/Power supply current <-> Data Pointer/PowerSupplyCurrent
//     Term 23 (APS4322-7000)/APS Inputs/StatusWord <-> Data Pointer/PowerUnitStatusWord
//     Term 23 (APS4322-7000)/APS Outputs/ControlWord <-> Data Pointer/PowerUnitControlWord
//     Term 23 (APS4322-7000)/APS Outputs/Current D 0X0 <-> Data Pointer/DCurrentSetPoints[0]
//     Term 23 (APS4322-7000)/APS Outputs/Current D 0X1 <-> Data Pointer/DCurrentSetPoints[1]
//     Term 23 (APS4322-7000)/APS Outputs/Current D 0X2 <-> Data Pointer/DCurrentSetPoints[2]
//     Term 23 (APS4322-7000)/APS Outputs/Current D 1X0 <-> Data Pointer/DCurrentSetPoints[6]
//     Term 23 (APS4322-7000)/APS Outputs/Current D 1X1 <-> Data Pointer/DCurrentSetPoints[7]
//     Term 23 (APS4322-7000)/APS Outputs/Current D 1X2 <-> Data Pointer/DCurrentSetPoints[8]
//     Term 23 (APS4322-7000)/APS Outputs/Current D 2X0 <-> Data Pointer/DCurrentSetPoints[12]
//     Term 23 (APS4322-7000)/APS Outputs/Current D 2X1 <-> Data Pointer/DCurrentSetPoints[13]
//     Term 23 (APS4322-7000)/APS Outputs/Current D 2X2 <-> Data Pointer/DCurrentSetPoints[14]
//     Term 23 (APS4322-7000)/APS Outputs/Current D 3X0 <-> Data Pointer/DCurrentSetPoints[18]
//     Term 23 (APS4322-7000)/APS Outputs/Current D 3X1 <-> Data Pointer/DCurrentSetPoints[19]
//     Term 23 (APS4322-7000)/APS Outputs/Current D 3X2 <-> Data Pointer/DCurrentSetPoints[20]
//     Term 23 (APS4322-7000)/APS Outputs/Current D 0Y0 <-> Data Pointer/DCurrentSetPoints[3]
//     Term 23 (APS4322-7000)/APS Outputs/Current D 0Y1 <-> Data Pointer/DCurrentSetPoints[4]
//     Term 23 (APS4322-7000)/APS Outputs/Current D 0Y2 <-> Data Pointer/DCurrentSetPoints[5]
//     Term 23 (APS4322-7000)/APS Outputs/Current D 1Y0 <-> Data Pointer/DCurrentSetPoints[9]
//     Term 23 (APS4322-7000)/APS Outputs/Current D 1Y1 <-> Data Pointer/DCurrentSetPoints[10]
//     Term 23 (APS4322-7000)/APS Outputs/Current D 1Y2 <-> Data Pointer/DCurrentSetPoints[11]
//     Term 23 (APS4322-7000)/APS Outputs/Current D 2Y0 <-> Data Pointer/DCurrentSetPoints[15]
//     Term 23 (APS4322-7000)/APS Outputs/Current D 2Y1 <-> Data Pointer/DCurrentSetPoints[16]
//     Term 23 (APS4322-7000)/APS Outputs/Current D 2Y2 <-> Data Pointer/DCurrentSetPoints[17]
//     Term 23 (APS4322-7000)/APS Outputs/Current D 3Y0 <-> Data Pointer/DCurrentSetPoints[21]
//     Term 23 (APS4322-7000)/APS Outputs/Current D 3Y1 <-> Data Pointer/DCurrentSetPoints[22]
//     Term 23 (APS4322-7000)/APS Outputs/Current D 3Y2 <-> Data Pointer/DCurrentSetPoints[23]
//     Term 23 (APS4322-7000)/APS Outputs/Current Q 0X0 <-> Data Pointer/QCurrentSetPoints[0]
//     Term 23 (APS4322-7000)/APS Outputs/Current Q 0X1 <-> Data Pointer/QCurrentSetPoints[1]
//     Term 23 (APS4322-7000)/APS Outputs/Current Q 0X2 <-> Data Pointer/QCurrentSetPoints[2]
//     Term 23 (APS4322-7000)/APS Outputs/Current Q 1X0 <-> Data Pointer/QCurrentSetPoints[6]
//     Term 23 (APS4322-7000)/APS Outputs/Current Q 1X1 <-> Data Pointer/QCurrentSetPoints[7]
//     Term 23 (APS4322-7000)/APS Outputs/Current Q 1X2 <-> Data Pointer/QCurrentSetPoints[8]
//     Term 23 (APS4322-7000)/APS Outputs/Current Q 2X0 <-> Data Pointer/QCurrentSetPoints[12]
//     Term 23 (APS4322-7000)/APS Outputs/Current Q 2X1 <-> Data Pointer/QCurrentSetPoints[13]
//     Term 23 (APS4322-7000)/APS Outputs/Current Q 2X2 <-> Data Pointer/QCurrentSetPoints[14]
//     Term 23 (APS4322-7000)/APS Outputs/Current Q 3X0 <-> Data Pointer/QCurrentSetPoints[18]
//     Term 23 (APS4322-7000)/APS Outputs/Current Q 3X1 <-> Data Pointer/QCurrentSetPoints[19]
//     Term 23 (APS4322-7000)/APS Outputs/Current Q 3X2 <-> Data Pointer/QCurrentSetPoints[20]
//     Term 23 (APS4322-7000)/APS Outputs/Current Q 0Y0 <-> Data Pointer/QCurrentSetPoints[3]
//     Term 23 (APS4322-7000)/APS Outputs/Current Q 0Y1 <-> Data Pointer/QCurrentSetPoints[4]
//     Term 23 (APS4322-7000)/APS Outputs/Current Q 0Y2 <-> Data Pointer/QCurrentSetPoints[5]
//     Term 23 (APS4322-7000)/APS Outputs/Current Q 1Y0 <-> Data Pointer/QCurrentSetPoints[9]
//     Term 23 (APS4322-7000)/APS Outputs/Current Q 1Y1 <-> Data Pointer/QCurrentSetPoints[10]
//     Term 23 (APS4322-7000)/APS Outputs/Current Q 1Y2 <-> Data Pointer/QCurrentSetPoints[11]
//     Term 23 (APS4322-7000)/APS Outputs/Current Q 2Y0 <-> Data Pointer/QCurrentSetPoints[15]
//     Term 23 (APS4322-7000)/APS Outputs/Current Q 2Y1 <-> Data Pointer/QCurrentSetPoints[16]
//     Term 23 (APS4322-7000)/APS Outputs/Current Q 2Y2 <-> Data Pointer/QCurrentSetPoints[17]
//     Term 23 (APS4322-7000)/APS Outputs/Current Q 3Y0 <-> Data Pointer/QCurrentSetPoints[21]
//     Term 23 (APS4322-7000)/APS Outputs/Current Q 3Y1 <-> Data Pointer/QCurrentSetPoints[22]
//     Term 23 (APS4322-7000)/APS Outputs/Current Q 3Y2 <-> Data Pointer/QCurrentSetPoints[23]
//     Term 23 (APS4322-7000)/APS Outputs/PhiE 0X0 <-> Data Pointer/PhiSetPoints[0]
//     Term 23 (APS4322-7000)/APS Outputs/PhiE 0X1 <-> Data Pointer/PhiSetPoints[1]
//     Term 23 (APS4322-7000)/APS Outputs/PhiE 0X2 <-> Data Pointer/PhiSetPoints[2]
//     Term 23 (APS4322-7000)/APS Outputs/PhiE 1X0 <-> Data Pointer/PhiSetPoints[6]
//     Term 23 (APS4322-7000)/APS Outputs/PhiE 1X1 <-> Data Pointer/PhiSetPoints[7]
//     Term 23 (APS4322-7000)/APS Outputs/PhiE 1X2 <-> Data Pointer/PhiSetPoints[8]
//     Term 23 (APS4322-7000)/APS Outputs/PhiE 2X0 <-> Data Pointer/PhiSetPoints[12]
//     Term 23 (APS4322-7000)/APS Outputs/PhiE 2X1 <-> Data Pointer/PhiSetPoints[13]
//     Term 23 (APS4322-7000)/APS Outputs/PhiE 2X2 <-> Data Pointer/PhiSetPoints[14]
//     Term 23 (APS4322-7000)/APS Outputs/PhiE 3X0 <-> Data Pointer/PhiSetPoints[18]
//     Term 23 (APS4322-7000)/APS Outputs/PhiE 3X1 <-> Data Pointer/PhiSetPoints[19]
//     Term 23 (APS4322-7000)/APS Outputs/PhiE 3X2 <-> Data Pointer/PhiSetPoints[20]
//     Term 23 (APS4322-7000)/APS Outputs/PhiE 0Y0 <-> Data Pointer/PhiSetPoints[3]
//     Term 23 (APS4322-7000)/APS Outputs/PhiE 0Y1 <-> Data Pointer/PhiSetPoints[4]
//     Term 23 (APS4322-7000)/APS Outputs/PhiE 0Y2 <-> Data Pointer/PhiSetPoints[5]
//     Term 23 (APS4322-7000)/APS Outputs/PhiE 1Y0 <-> Data Pointer/PhiSetPoints[9]
//     Term 23 (APS4322-7000)/APS Outputs/PhiE 1Y1 <-> Data Pointer/PhiSetPoints[10]
//     Term 23 (APS4322-7000)/APS Outputs/PhiE 1Y2 <-> Data Pointer/PhiSetPoints[11]
//     Term 23 (APS4322-7000)/APS Outputs/PhiE 2Y0 <-> Data Pointer/PhiSetPoints[15]
//     Term 23 (APS4322-7000)/APS Outputs/PhiE 2Y1 <-> Data Pointer/PhiSetPoints[16]
//     Term 23 (APS4322-7000)/APS Outputs/PhiE 2Y2 <-> Data Pointer/PhiSetPoints[17]
//     Term 23 (APS4322-7000)/APS Outputs/PhiE 3Y0 <-> Data Pointer/PhiSetPoints[21]
//     Term 23 (APS4322-7000)/APS Outputs/PhiE 3Y1 <-> Data Pointer/PhiSetPoints[22]
//     Term 23 (APS4322-7000)/APS Outputs/PhiE 3Y2 <-> Data Pointer/PhiSetPoints[23]
//     Term 23 (APS4322-7000)/Term 24 (APS4322-5000)/FB Inputs/A{0..8 step 2} X-Field <-> Data Pointer/HallSensorFieldsXYZ[{0..12 step 3}]  (5 links)
//     Term 23 (APS4322-7000)/Term 24 (APS4322-5000)/FB Inputs/A{0..8 step 2} Y-Field <-> Data Pointer/HallSensorFieldsXYZ[{1..13 step 3}]  (5 links)
//     Term 23 (APS4322-7000)/Term 24 (APS4322-5000)/FB Inputs/A{0..8 step 2} Z-Field <-> Data Pointer/HallSensorFieldsXYZ[{2..14 step 3}]  (5 links)
//     Term 23 (APS4322-7000)/Term 24 (APS4322-5000)/FB Inputs/B{1..9 step 2} X-Field <-> Data Pointer/HallSensorFieldsXYZ[{15..27 step 3}]  (5 links)
//     Term 23 (APS4322-7000)/Term 24 (APS4322-5000)/FB Inputs/B{1..9 step 2} Y-Field <-> Data Pointer/HallSensorFieldsXYZ[{16..28 step 3}]  (5 links)
//     Term 23 (APS4322-7000)/Term 24 (APS4322-5000)/FB Inputs/B{1..9 step 2} Z-Field <-> Data Pointer/HallSensorFieldsXYZ[{17..29 step 3}]  (5 links)
//     Term 23 (APS4322-7000)/Term 24 (APS4322-5000)/FB Inputs/C{0..8 step 2} X-Field <-> Data Pointer/HallSensorFieldsXYZ[{30..42 step 3}]  (5 links)
//     Term 23 (APS4322-7000)/Term 24 (APS4322-5000)/FB Inputs/C{0..8 step 2} Y-Field <-> Data Pointer/HallSensorFieldsXYZ[{31..43 step 3}]  (5 links)
//     Term 23 (APS4322-7000)/Term 24 (APS4322-5000)/FB Inputs/C{0..8 step 2} Z-Field <-> Data Pointer/HallSensorFieldsXYZ[{32..44 step 3}]  (5 links)
//     Term 23 (APS4322-7000)/Term 24 (APS4322-5000)/FB Inputs/D{1..9 step 2} X-Field <-> Data Pointer/HallSensorFieldsXYZ[{45..57 step 3}]  (5 links)
//     Term 23 (APS4322-7000)/Term 24 (APS4322-5000)/FB Inputs/D{1..9 step 2} Y-Field <-> Data Pointer/HallSensorFieldsXYZ[{46..58 step 3}]  (5 links)
//     Term 23 (APS4322-7000)/Term 24 (APS4322-5000)/FB Inputs/D{1..9 step 2} Z-Field <-> Data Pointer/HallSensorFieldsXYZ[{47..59 step 3}]  (5 links)
//     Term 23 (APS4322-7000)/Term 24 (APS4322-5000)/FB Inputs/E{0..8 step 2} X-Field <-> Data Pointer/HallSensorFieldsXYZ[{60..72 step 3}]  (5 links)
//     Term 23 (APS4322-7000)/Term 24 (APS4322-5000)/FB Inputs/E{0..8 step 2} Y-Field <-> Data Pointer/HallSensorFieldsXYZ[{61..73 step 3}]  (5 links)
//     Term 23 (APS4322-7000)/Term 24 (APS4322-5000)/FB Inputs/E{0..8 step 2} Z-Field <-> Data Pointer/HallSensorFieldsXYZ[{62..74 step 3}]  (5 links)
//     Term 23 (APS4322-7000)/Term 24 (APS4322-5000)/FB Inputs/F{1..9 step 2} X-Field <-> Data Pointer/HallSensorFieldsXYZ[{75..87 step 3}]  (5 links)
//     Term 23 (APS4322-7000)/Term 24 (APS4322-5000)/FB Inputs/F{1..9 step 2} Y-Field <-> Data Pointer/HallSensorFieldsXYZ[{76..88 step 3}]  (5 links)
//     Term 23 (APS4322-7000)/Term 24 (APS4322-5000)/FB Inputs/F{1..9 step 2} Z-Field <-> Data Pointer/HallSensorFieldsXYZ[{77..89 step 3}]  (5 links)
//     Term 23 (APS4322-7000)/Term 24 (APS4322-5000)/FB Inputs/G{0..8 step 2} X-Field <-> Data Pointer/HallSensorFieldsXYZ[{90..102 step 3}]  (5 links)
//     Term 23 (APS4322-7000)/Term 24 (APS4322-5000)/FB Inputs/G{0..8 step 2} Y-Field <-> Data Pointer/HallSensorFieldsXYZ[{91..103 step 3}]  (5 links)
//     Term 23 (APS4322-7000)/Term 24 (APS4322-5000)/FB Inputs/G{0..8 step 2} Z-Field <-> Data Pointer/HallSensorFieldsXYZ[{92..104 step 3}]  (5 links)
//     Term 23 (APS4322-7000)/Term 24 (APS4322-5000)/FB Inputs/H{1..9 step 2} X-Field <-> Data Pointer/HallSensorFieldsXYZ[{105..117 step 3}]  (5 links)
//     Term 23 (APS4322-7000)/Term 24 (APS4322-5000)/FB Inputs/H{1..9 step 2} Y-Field <-> Data Pointer/HallSensorFieldsXYZ[{106..118 step 3}]  (5 links)
//     Term 23 (APS4322-7000)/Term 24 (APS4322-5000)/FB Inputs/H{1..9 step 2} Z-Field <-> Data Pointer/HallSensorFieldsXYZ[{107..119 step 3}]  (5 links)
//     Term 23 (APS4322-7000)/Term 24 (APS4322-5000)/FB Inputs/I{0..8 step 2} X-Field <-> Data Pointer/HallSensorFieldsXYZ[{120..132 step 3}]  (5 links)
//     Term 23 (APS4322-7000)/Term 24 (APS4322-5000)/FB Inputs/I{0..8 step 2} Y-Field <-> Data Pointer/HallSensorFieldsXYZ[{121..133 step 3}]  (5 links)
//     Term 23 (APS4322-7000)/Term 24 (APS4322-5000)/FB Inputs/I{0..8 step 2} Z-Field <-> Data Pointer/HallSensorFieldsXYZ[{122..134 step 3}]  (5 links)
//     Term 23 (APS4322-7000)/Term 24 (APS4322-5000)/FB Inputs/J{1..9 step 2} X-Field <-> Data Pointer/HallSensorFieldsXYZ[{135..147 step 3}]  (5 links)
//     Term 23 (APS4322-7000)/Term 24 (APS4322-5000)/FB Inputs/J{1..9 step 2} Y-Field <-> Data Pointer/HallSensorFieldsXYZ[{136..148 step 3}]  (5 links)
//     Term 23 (APS4322-7000)/Term 24 (APS4322-5000)/FB Inputs/J{1..9 step 2} Z-Field <-> Data Pointer/HallSensorFieldsXYZ[{137..149 step 3}]  (5 links)
//     Term 23 (APS4322-7000)/Term 24 (APS4322-5000)/FB Inputs/Status <-> Data Pointer/FeedbackStatus
//   Device 2 (EtherCAT) <-> TcCOM Objects/XPlanar/Part1/Tile9
//     Term 25 (APS4322-7000)/APS Comm Inputs/CommStatusWord <-> Data Pointer/MoverCommStatusWord
//     Term 25 (APS4322-7000)/APS Comm Inputs/Data {1..4} <-> Data Pointer/MoverCommDataIn[{0..3}]  (4 links)
//     Term 25 (APS4322-7000)/APS Comm Outputs/CommControlWord <-> Data Pointer/MoverCommControlWord
//     Term 25 (APS4322-7000)/APS Comm Outputs/Data 1 <-> Data Pointer/MoverCommDataOut
//     Term 25 (APS4322-7000)/APS Diagdata/DC Link Voltage <-> Data Pointer/DcLinkVoltage
//     Term 25 (APS4322-7000)/APS Diagdata/Power supply current <-> Data Pointer/PowerSupplyCurrent
//     Term 25 (APS4322-7000)/APS Inputs/StatusWord <-> Data Pointer/PowerUnitStatusWord
//     Term 25 (APS4322-7000)/APS Outputs/ControlWord <-> Data Pointer/PowerUnitControlWord
//     Term 25 (APS4322-7000)/APS Outputs/Current D 0X0 <-> Data Pointer/DCurrentSetPoints[0]
//     Term 25 (APS4322-7000)/APS Outputs/Current D 0X1 <-> Data Pointer/DCurrentSetPoints[1]
//     Term 25 (APS4322-7000)/APS Outputs/Current D 0X2 <-> Data Pointer/DCurrentSetPoints[2]
//     Term 25 (APS4322-7000)/APS Outputs/Current D 1X0 <-> Data Pointer/DCurrentSetPoints[6]
//     Term 25 (APS4322-7000)/APS Outputs/Current D 1X1 <-> Data Pointer/DCurrentSetPoints[7]
//     Term 25 (APS4322-7000)/APS Outputs/Current D 1X2 <-> Data Pointer/DCurrentSetPoints[8]
//     Term 25 (APS4322-7000)/APS Outputs/Current D 2X0 <-> Data Pointer/DCurrentSetPoints[12]
//     Term 25 (APS4322-7000)/APS Outputs/Current D 2X1 <-> Data Pointer/DCurrentSetPoints[13]
//     Term 25 (APS4322-7000)/APS Outputs/Current D 2X2 <-> Data Pointer/DCurrentSetPoints[14]
//     Term 25 (APS4322-7000)/APS Outputs/Current D 3X0 <-> Data Pointer/DCurrentSetPoints[18]
//     Term 25 (APS4322-7000)/APS Outputs/Current D 3X1 <-> Data Pointer/DCurrentSetPoints[19]
//     Term 25 (APS4322-7000)/APS Outputs/Current D 3X2 <-> Data Pointer/DCurrentSetPoints[20]
//     Term 25 (APS4322-7000)/APS Outputs/Current D 0Y0 <-> Data Pointer/DCurrentSetPoints[3]
//     Term 25 (APS4322-7000)/APS Outputs/Current D 0Y1 <-> Data Pointer/DCurrentSetPoints[4]
//     Term 25 (APS4322-7000)/APS Outputs/Current D 0Y2 <-> Data Pointer/DCurrentSetPoints[5]
//     Term 25 (APS4322-7000)/APS Outputs/Current D 1Y0 <-> Data Pointer/DCurrentSetPoints[9]
//     Term 25 (APS4322-7000)/APS Outputs/Current D 1Y1 <-> Data Pointer/DCurrentSetPoints[10]
//     Term 25 (APS4322-7000)/APS Outputs/Current D 1Y2 <-> Data Pointer/DCurrentSetPoints[11]
//     Term 25 (APS4322-7000)/APS Outputs/Current D 2Y0 <-> Data Pointer/DCurrentSetPoints[15]
//     Term 25 (APS4322-7000)/APS Outputs/Current D 2Y1 <-> Data Pointer/DCurrentSetPoints[16]
//     Term 25 (APS4322-7000)/APS Outputs/Current D 2Y2 <-> Data Pointer/DCurrentSetPoints[17]
//     Term 25 (APS4322-7000)/APS Outputs/Current D 3Y0 <-> Data Pointer/DCurrentSetPoints[21]
//     Term 25 (APS4322-7000)/APS Outputs/Current D 3Y1 <-> Data Pointer/DCurrentSetPoints[22]
//     Term 25 (APS4322-7000)/APS Outputs/Current D 3Y2 <-> Data Pointer/DCurrentSetPoints[23]
//     Term 25 (APS4322-7000)/APS Outputs/Current Q 0X0 <-> Data Pointer/QCurrentSetPoints[0]
//     Term 25 (APS4322-7000)/APS Outputs/Current Q 0X1 <-> Data Pointer/QCurrentSetPoints[1]
//     Term 25 (APS4322-7000)/APS Outputs/Current Q 0X2 <-> Data Pointer/QCurrentSetPoints[2]
//     Term 25 (APS4322-7000)/APS Outputs/Current Q 1X0 <-> Data Pointer/QCurrentSetPoints[6]
//     Term 25 (APS4322-7000)/APS Outputs/Current Q 1X1 <-> Data Pointer/QCurrentSetPoints[7]
//     Term 25 (APS4322-7000)/APS Outputs/Current Q 1X2 <-> Data Pointer/QCurrentSetPoints[8]
//     Term 25 (APS4322-7000)/APS Outputs/Current Q 2X0 <-> Data Pointer/QCurrentSetPoints[12]
//     Term 25 (APS4322-7000)/APS Outputs/Current Q 2X1 <-> Data Pointer/QCurrentSetPoints[13]
//     Term 25 (APS4322-7000)/APS Outputs/Current Q 2X2 <-> Data Pointer/QCurrentSetPoints[14]
//     Term 25 (APS4322-7000)/APS Outputs/Current Q 3X0 <-> Data Pointer/QCurrentSetPoints[18]
//     Term 25 (APS4322-7000)/APS Outputs/Current Q 3X1 <-> Data Pointer/QCurrentSetPoints[19]
//     Term 25 (APS4322-7000)/APS Outputs/Current Q 3X2 <-> Data Pointer/QCurrentSetPoints[20]
//     Term 25 (APS4322-7000)/APS Outputs/Current Q 0Y0 <-> Data Pointer/QCurrentSetPoints[3]
//     Term 25 (APS4322-7000)/APS Outputs/Current Q 0Y1 <-> Data Pointer/QCurrentSetPoints[4]
//     Term 25 (APS4322-7000)/APS Outputs/Current Q 0Y2 <-> Data Pointer/QCurrentSetPoints[5]
//     Term 25 (APS4322-7000)/APS Outputs/Current Q 1Y0 <-> Data Pointer/QCurrentSetPoints[9]
//     Term 25 (APS4322-7000)/APS Outputs/Current Q 1Y1 <-> Data Pointer/QCurrentSetPoints[10]
//     Term 25 (APS4322-7000)/APS Outputs/Current Q 1Y2 <-> Data Pointer/QCurrentSetPoints[11]
//     Term 25 (APS4322-7000)/APS Outputs/Current Q 2Y0 <-> Data Pointer/QCurrentSetPoints[15]
//     Term 25 (APS4322-7000)/APS Outputs/Current Q 2Y1 <-> Data Pointer/QCurrentSetPoints[16]
//     Term 25 (APS4322-7000)/APS Outputs/Current Q 2Y2 <-> Data Pointer/QCurrentSetPoints[17]
//     Term 25 (APS4322-7000)/APS Outputs/Current Q 3Y0 <-> Data Pointer/QCurrentSetPoints[21]
//     Term 25 (APS4322-7000)/APS Outputs/Current Q 3Y1 <-> Data Pointer/QCurrentSetPoints[22]
//     Term 25 (APS4322-7000)/APS Outputs/Current Q 3Y2 <-> Data Pointer/QCurrentSetPoints[23]
//     Term 25 (APS4322-7000)/APS Outputs/PhiE 0X0 <-> Data Pointer/PhiSetPoints[0]
//     Term 25 (APS4322-7000)/APS Outputs/PhiE 0X1 <-> Data Pointer/PhiSetPoints[1]
//     Term 25 (APS4322-7000)/APS Outputs/PhiE 0X2 <-> Data Pointer/PhiSetPoints[2]
//     Term 25 (APS4322-7000)/APS Outputs/PhiE 1X0 <-> Data Pointer/PhiSetPoints[6]
//     Term 25 (APS4322-7000)/APS Outputs/PhiE 1X1 <-> Data Pointer/PhiSetPoints[7]
//     Term 25 (APS4322-7000)/APS Outputs/PhiE 1X2 <-> Data Pointer/PhiSetPoints[8]
//     Term 25 (APS4322-7000)/APS Outputs/PhiE 2X0 <-> Data Pointer/PhiSetPoints[12]
//     Term 25 (APS4322-7000)/APS Outputs/PhiE 2X1 <-> Data Pointer/PhiSetPoints[13]
//     Term 25 (APS4322-7000)/APS Outputs/PhiE 2X2 <-> Data Pointer/PhiSetPoints[14]
//     Term 25 (APS4322-7000)/APS Outputs/PhiE 3X0 <-> Data Pointer/PhiSetPoints[18]
//     Term 25 (APS4322-7000)/APS Outputs/PhiE 3X1 <-> Data Pointer/PhiSetPoints[19]
//     Term 25 (APS4322-7000)/APS Outputs/PhiE 3X2 <-> Data Pointer/PhiSetPoints[20]
//     Term 25 (APS4322-7000)/APS Outputs/PhiE 0Y0 <-> Data Pointer/PhiSetPoints[3]
//     Term 25 (APS4322-7000)/APS Outputs/PhiE 0Y1 <-> Data Pointer/PhiSetPoints[4]
//     Term 25 (APS4322-7000)/APS Outputs/PhiE 0Y2 <-> Data Pointer/PhiSetPoints[5]
//     Term 25 (APS4322-7000)/APS Outputs/PhiE 1Y0 <-> Data Pointer/PhiSetPoints[9]
//     Term 25 (APS4322-7000)/APS Outputs/PhiE 1Y1 <-> Data Pointer/PhiSetPoints[10]
//     Term 25 (APS4322-7000)/APS Outputs/PhiE 1Y2 <-> Data Pointer/PhiSetPoints[11]
//     Term 25 (APS4322-7000)/APS Outputs/PhiE 2Y0 <-> Data Pointer/PhiSetPoints[15]
//     Term 25 (APS4322-7000)/APS Outputs/PhiE 2Y1 <-> Data Pointer/PhiSetPoints[16]
//     Term 25 (APS4322-7000)/APS Outputs/PhiE 2Y2 <-> Data Pointer/PhiSetPoints[17]
//     Term 25 (APS4322-7000)/APS Outputs/PhiE 3Y0 <-> Data Pointer/PhiSetPoints[21]
//     Term 25 (APS4322-7000)/APS Outputs/PhiE 3Y1 <-> Data Pointer/PhiSetPoints[22]
//     Term 25 (APS4322-7000)/APS Outputs/PhiE 3Y2 <-> Data Pointer/PhiSetPoints[23]
//     Term 25 (APS4322-7000)/Term 26 (APS4322-5000)/FB Inputs/A{0..8 step 2} X-Field <-> Data Pointer/HallSensorFieldsXYZ[{0..12 step 3}]  (5 links)
//     Term 25 (APS4322-7000)/Term 26 (APS4322-5000)/FB Inputs/A{0..8 step 2} Y-Field <-> Data Pointer/HallSensorFieldsXYZ[{1..13 step 3}]  (5 links)
//     Term 25 (APS4322-7000)/Term 26 (APS4322-5000)/FB Inputs/A{0..8 step 2} Z-Field <-> Data Pointer/HallSensorFieldsXYZ[{2..14 step 3}]  (5 links)
//     Term 25 (APS4322-7000)/Term 26 (APS4322-5000)/FB Inputs/B{1..9 step 2} X-Field <-> Data Pointer/HallSensorFieldsXYZ[{15..27 step 3}]  (5 links)
//     Term 25 (APS4322-7000)/Term 26 (APS4322-5000)/FB Inputs/B{1..9 step 2} Y-Field <-> Data Pointer/HallSensorFieldsXYZ[{16..28 step 3}]  (5 links)
//     Term 25 (APS4322-7000)/Term 26 (APS4322-5000)/FB Inputs/B{1..9 step 2} Z-Field <-> Data Pointer/HallSensorFieldsXYZ[{17..29 step 3}]  (5 links)
//     Term 25 (APS4322-7000)/Term 26 (APS4322-5000)/FB Inputs/C{0..8 step 2} X-Field <-> Data Pointer/HallSensorFieldsXYZ[{30..42 step 3}]  (5 links)
//     Term 25 (APS4322-7000)/Term 26 (APS4322-5000)/FB Inputs/C{0..8 step 2} Y-Field <-> Data Pointer/HallSensorFieldsXYZ[{31..43 step 3}]  (5 links)
//     Term 25 (APS4322-7000)/Term 26 (APS4322-5000)/FB Inputs/C{0..8 step 2} Z-Field <-> Data Pointer/HallSensorFieldsXYZ[{32..44 step 3}]  (5 links)
//     Term 25 (APS4322-7000)/Term 26 (APS4322-5000)/FB Inputs/D{1..9 step 2} X-Field <-> Data Pointer/HallSensorFieldsXYZ[{45..57 step 3}]  (5 links)
//     Term 25 (APS4322-7000)/Term 26 (APS4322-5000)/FB Inputs/D{1..9 step 2} Y-Field <-> Data Pointer/HallSensorFieldsXYZ[{46..58 step 3}]  (5 links)
//     Term 25 (APS4322-7000)/Term 26 (APS4322-5000)/FB Inputs/D{1..9 step 2} Z-Field <-> Data Pointer/HallSensorFieldsXYZ[{47..59 step 3}]  (5 links)
//     Term 25 (APS4322-7000)/Term 26 (APS4322-5000)/FB Inputs/E{0..8 step 2} X-Field <-> Data Pointer/HallSensorFieldsXYZ[{60..72 step 3}]  (5 links)
//     Term 25 (APS4322-7000)/Term 26 (APS4322-5000)/FB Inputs/E{0..8 step 2} Y-Field <-> Data Pointer/HallSensorFieldsXYZ[{61..73 step 3}]  (5 links)
//     Term 25 (APS4322-7000)/Term 26 (APS4322-5000)/FB Inputs/E{0..8 step 2} Z-Field <-> Data Pointer/HallSensorFieldsXYZ[{62..74 step 3}]  (5 links)
//     Term 25 (APS4322-7000)/Term 26 (APS4322-5000)/FB Inputs/F{1..9 step 2} X-Field <-> Data Pointer/HallSensorFieldsXYZ[{75..87 step 3}]  (5 links)
//     Term 25 (APS4322-7000)/Term 26 (APS4322-5000)/FB Inputs/F{1..9 step 2} Y-Field <-> Data Pointer/HallSensorFieldsXYZ[{76..88 step 3}]  (5 links)
//     Term 25 (APS4322-7000)/Term 26 (APS4322-5000)/FB Inputs/F{1..9 step 2} Z-Field <-> Data Pointer/HallSensorFieldsXYZ[{77..89 step 3}]  (5 links)
//     Term 25 (APS4322-7000)/Term 26 (APS4322-5000)/FB Inputs/G{0..8 step 2} X-Field <-> Data Pointer/HallSensorFieldsXYZ[{90..102 step 3}]  (5 links)
//     Term 25 (APS4322-7000)/Term 26 (APS4322-5000)/FB Inputs/G{0..8 step 2} Y-Field <-> Data Pointer/HallSensorFieldsXYZ[{91..103 step 3}]  (5 links)
//     Term 25 (APS4322-7000)/Term 26 (APS4322-5000)/FB Inputs/G{0..8 step 2} Z-Field <-> Data Pointer/HallSensorFieldsXYZ[{92..104 step 3}]  (5 links)
//     Term 25 (APS4322-7000)/Term 26 (APS4322-5000)/FB Inputs/H{1..9 step 2} X-Field <-> Data Pointer/HallSensorFieldsXYZ[{105..117 step 3}]  (5 links)
//     Term 25 (APS4322-7000)/Term 26 (APS4322-5000)/FB Inputs/H{1..9 step 2} Y-Field <-> Data Pointer/HallSensorFieldsXYZ[{106..118 step 3}]  (5 links)
//     Term 25 (APS4322-7000)/Term 26 (APS4322-5000)/FB Inputs/H{1..9 step 2} Z-Field <-> Data Pointer/HallSensorFieldsXYZ[{107..119 step 3}]  (5 links)
//     Term 25 (APS4322-7000)/Term 26 (APS4322-5000)/FB Inputs/I{0..8 step 2} X-Field <-> Data Pointer/HallSensorFieldsXYZ[{120..132 step 3}]  (5 links)
//     Term 25 (APS4322-7000)/Term 26 (APS4322-5000)/FB Inputs/I{0..8 step 2} Y-Field <-> Data Pointer/HallSensorFieldsXYZ[{121..133 step 3}]  (5 links)
//     Term 25 (APS4322-7000)/Term 26 (APS4322-5000)/FB Inputs/I{0..8 step 2} Z-Field <-> Data Pointer/HallSensorFieldsXYZ[{122..134 step 3}]  (5 links)
//     Term 25 (APS4322-7000)/Term 26 (APS4322-5000)/FB Inputs/J{1..9 step 2} X-Field <-> Data Pointer/HallSensorFieldsXYZ[{135..147 step 3}]  (5 links)
//     Term 25 (APS4322-7000)/Term 26 (APS4322-5000)/FB Inputs/J{1..9 step 2} Y-Field <-> Data Pointer/HallSensorFieldsXYZ[{136..148 step 3}]  (5 links)
//     Term 25 (APS4322-7000)/Term 26 (APS4322-5000)/FB Inputs/J{1..9 step 2} Z-Field <-> Data Pointer/HallSensorFieldsXYZ[{137..149 step 3}]  (5 links)
//     Term 25 (APS4322-7000)/Term 26 (APS4322-5000)/FB Inputs/Status <-> Data Pointer/FeedbackStatus
//   Device 6 (EtherCAT) <-> TcCOM Objects/XPlanar/Part1/Tile11
//     Term 13 (APS4322-7000)/APS Comm Inputs/CommStatusWord <-> Data Pointer/MoverCommStatusWord
//     Term 13 (APS4322-7000)/APS Comm Inputs/Data {1..4} <-> Data Pointer/MoverCommDataIn[{0..3}]  (4 links)
//     Term 13 (APS4322-7000)/APS Comm Outputs/CommControlWord <-> Data Pointer/MoverCommControlWord
//     Term 13 (APS4322-7000)/APS Comm Outputs/Data 1 <-> Data Pointer/MoverCommDataOut
//     Term 13 (APS4322-7000)/APS Diagdata/DC Link Voltage <-> Data Pointer/DcLinkVoltage
//     Term 13 (APS4322-7000)/APS Diagdata/Power supply current <-> Data Pointer/PowerSupplyCurrent
//     Term 13 (APS4322-7000)/APS Inputs/StatusWord <-> Data Pointer/PowerUnitStatusWord
//     Term 13 (APS4322-7000)/APS Outputs/ControlWord <-> Data Pointer/PowerUnitControlWord
//     Term 13 (APS4322-7000)/APS Outputs/Current D 0X0 <-> Data Pointer/DCurrentSetPoints[0]
//     Term 13 (APS4322-7000)/APS Outputs/Current D 0X1 <-> Data Pointer/DCurrentSetPoints[1]
//     Term 13 (APS4322-7000)/APS Outputs/Current D 0X2 <-> Data Pointer/DCurrentSetPoints[2]
//     Term 13 (APS4322-7000)/APS Outputs/Current D 1X0 <-> Data Pointer/DCurrentSetPoints[6]
//     Term 13 (APS4322-7000)/APS Outputs/Current D 1X1 <-> Data Pointer/DCurrentSetPoints[7]
//     Term 13 (APS4322-7000)/APS Outputs/Current D 1X2 <-> Data Pointer/DCurrentSetPoints[8]
//     Term 13 (APS4322-7000)/APS Outputs/Current D 2X0 <-> Data Pointer/DCurrentSetPoints[12]
//     Term 13 (APS4322-7000)/APS Outputs/Current D 2X1 <-> Data Pointer/DCurrentSetPoints[13]
//     Term 13 (APS4322-7000)/APS Outputs/Current D 2X2 <-> Data Pointer/DCurrentSetPoints[14]
//     Term 13 (APS4322-7000)/APS Outputs/Current D 3X0 <-> Data Pointer/DCurrentSetPoints[18]
//     Term 13 (APS4322-7000)/APS Outputs/Current D 3X1 <-> Data Pointer/DCurrentSetPoints[19]
//     Term 13 (APS4322-7000)/APS Outputs/Current D 3X2 <-> Data Pointer/DCurrentSetPoints[20]
//     Term 13 (APS4322-7000)/APS Outputs/Current D 0Y0 <-> Data Pointer/DCurrentSetPoints[3]
//     Term 13 (APS4322-7000)/APS Outputs/Current D 0Y1 <-> Data Pointer/DCurrentSetPoints[4]
//     Term 13 (APS4322-7000)/APS Outputs/Current D 0Y2 <-> Data Pointer/DCurrentSetPoints[5]
//     Term 13 (APS4322-7000)/APS Outputs/Current D 1Y0 <-> Data Pointer/DCurrentSetPoints[9]
//     Term 13 (APS4322-7000)/APS Outputs/Current D 1Y1 <-> Data Pointer/DCurrentSetPoints[10]
//     Term 13 (APS4322-7000)/APS Outputs/Current D 1Y2 <-> Data Pointer/DCurrentSetPoints[11]
//     Term 13 (APS4322-7000)/APS Outputs/Current D 2Y0 <-> Data Pointer/DCurrentSetPoints[15]
//     Term 13 (APS4322-7000)/APS Outputs/Current D 2Y1 <-> Data Pointer/DCurrentSetPoints[16]
//     Term 13 (APS4322-7000)/APS Outputs/Current D 2Y2 <-> Data Pointer/DCurrentSetPoints[17]
//     Term 13 (APS4322-7000)/APS Outputs/Current D 3Y0 <-> Data Pointer/DCurrentSetPoints[21]
//     Term 13 (APS4322-7000)/APS Outputs/Current D 3Y1 <-> Data Pointer/DCurrentSetPoints[22]
//     Term 13 (APS4322-7000)/APS Outputs/Current D 3Y2 <-> Data Pointer/DCurrentSetPoints[23]
//     Term 13 (APS4322-7000)/APS Outputs/Current Q 0X0 <-> Data Pointer/QCurrentSetPoints[0]
//     Term 13 (APS4322-7000)/APS Outputs/Current Q 0X1 <-> Data Pointer/QCurrentSetPoints[1]
//     Term 13 (APS4322-7000)/APS Outputs/Current Q 0X2 <-> Data Pointer/QCurrentSetPoints[2]
//     Term 13 (APS4322-7000)/APS Outputs/Current Q 1X0 <-> Data Pointer/QCurrentSetPoints[6]
//     Term 13 (APS4322-7000)/APS Outputs/Current Q 1X1 <-> Data Pointer/QCurrentSetPoints[7]
//     Term 13 (APS4322-7000)/APS Outputs/Current Q 1X2 <-> Data Pointer/QCurrentSetPoints[8]
//     Term 13 (APS4322-7000)/APS Outputs/Current Q 2X0 <-> Data Pointer/QCurrentSetPoints[12]
//     Term 13 (APS4322-7000)/APS Outputs/Current Q 2X1 <-> Data Pointer/QCurrentSetPoints[13]
//     Term 13 (APS4322-7000)/APS Outputs/Current Q 2X2 <-> Data Pointer/QCurrentSetPoints[14]
//     Term 13 (APS4322-7000)/APS Outputs/Current Q 3X0 <-> Data Pointer/QCurrentSetPoints[18]
//     Term 13 (APS4322-7000)/APS Outputs/Current Q 3X1 <-> Data Pointer/QCurrentSetPoints[19]
//     Term 13 (APS4322-7000)/APS Outputs/Current Q 3X2 <-> Data Pointer/QCurrentSetPoints[20]
//     Term 13 (APS4322-7000)/APS Outputs/Current Q 0Y0 <-> Data Pointer/QCurrentSetPoints[3]
//     Term 13 (APS4322-7000)/APS Outputs/Current Q 0Y1 <-> Data Pointer/QCurrentSetPoints[4]
//     Term 13 (APS4322-7000)/APS Outputs/Current Q 0Y2 <-> Data Pointer/QCurrentSetPoints[5]
//     Term 13 (APS4322-7000)/APS Outputs/Current Q 1Y0 <-> Data Pointer/QCurrentSetPoints[9]
//     Term 13 (APS4322-7000)/APS Outputs/Current Q 1Y1 <-> Data Pointer/QCurrentSetPoints[10]
//     Term 13 (APS4322-7000)/APS Outputs/Current Q 1Y2 <-> Data Pointer/QCurrentSetPoints[11]
//     Term 13 (APS4322-7000)/APS Outputs/Current Q 2Y0 <-> Data Pointer/QCurrentSetPoints[15]
//     Term 13 (APS4322-7000)/APS Outputs/Current Q 2Y1 <-> Data Pointer/QCurrentSetPoints[16]
//     Term 13 (APS4322-7000)/APS Outputs/Current Q 2Y2 <-> Data Pointer/QCurrentSetPoints[17]
//     Term 13 (APS4322-7000)/APS Outputs/Current Q 3Y0 <-> Data Pointer/QCurrentSetPoints[21]
//     Term 13 (APS4322-7000)/APS Outputs/Current Q 3Y1 <-> Data Pointer/QCurrentSetPoints[22]
//     Term 13 (APS4322-7000)/APS Outputs/Current Q 3Y2 <-> Data Pointer/QCurrentSetPoints[23]
//     Term 13 (APS4322-7000)/APS Outputs/PhiE 0X0 <-> Data Pointer/PhiSetPoints[0]
//     Term 13 (APS4322-7000)/APS Outputs/PhiE 0X1 <-> Data Pointer/PhiSetPoints[1]
//     Term 13 (APS4322-7000)/APS Outputs/PhiE 0X2 <-> Data Pointer/PhiSetPoints[2]
//     Term 13 (APS4322-7000)/APS Outputs/PhiE 1X0 <-> Data Pointer/PhiSetPoints[6]
//     Term 13 (APS4322-7000)/APS Outputs/PhiE 1X1 <-> Data Pointer/PhiSetPoints[7]
//     Term 13 (APS4322-7000)/APS Outputs/PhiE 1X2 <-> Data Pointer/PhiSetPoints[8]
//     Term 13 (APS4322-7000)/APS Outputs/PhiE 2X0 <-> Data Pointer/PhiSetPoints[12]
//     Term 13 (APS4322-7000)/APS Outputs/PhiE 2X1 <-> Data Pointer/PhiSetPoints[13]
//     Term 13 (APS4322-7000)/APS Outputs/PhiE 2X2 <-> Data Pointer/PhiSetPoints[14]
//     Term 13 (APS4322-7000)/APS Outputs/PhiE 3X0 <-> Data Pointer/PhiSetPoints[18]
//     Term 13 (APS4322-7000)/APS Outputs/PhiE 3X1 <-> Data Pointer/PhiSetPoints[19]
//     Term 13 (APS4322-7000)/APS Outputs/PhiE 3X2 <-> Data Pointer/PhiSetPoints[20]
//     Term 13 (APS4322-7000)/APS Outputs/PhiE 0Y0 <-> Data Pointer/PhiSetPoints[3]
//     Term 13 (APS4322-7000)/APS Outputs/PhiE 0Y1 <-> Data Pointer/PhiSetPoints[4]
//     Term 13 (APS4322-7000)/APS Outputs/PhiE 0Y2 <-> Data Pointer/PhiSetPoints[5]
//     Term 13 (APS4322-7000)/APS Outputs/PhiE 1Y0 <-> Data Pointer/PhiSetPoints[9]
//     Term 13 (APS4322-7000)/APS Outputs/PhiE 1Y1 <-> Data Pointer/PhiSetPoints[10]
//     Term 13 (APS4322-7000)/APS Outputs/PhiE 1Y2 <-> Data Pointer/PhiSetPoints[11]
//     Term 13 (APS4322-7000)/APS Outputs/PhiE 2Y0 <-> Data Pointer/PhiSetPoints[15]
//     Term 13 (APS4322-7000)/APS Outputs/PhiE 2Y1 <-> Data Pointer/PhiSetPoints[16]
//     Term 13 (APS4322-7000)/APS Outputs/PhiE 2Y2 <-> Data Pointer/PhiSetPoints[17]
//     Term 13 (APS4322-7000)/APS Outputs/PhiE 3Y0 <-> Data Pointer/PhiSetPoints[21]
//     Term 13 (APS4322-7000)/APS Outputs/PhiE 3Y1 <-> Data Pointer/PhiSetPoints[22]
//     Term 13 (APS4322-7000)/APS Outputs/PhiE 3Y2 <-> Data Pointer/PhiSetPoints[23]
//     Term 13 (APS4322-7000)/Term 14 (APS4322-5000)/FB Inputs/A{0..8 step 2} X-Field <-> Data Pointer/HallSensorFieldsXYZ[{0..12 step 3}]  (5 links)
//     Term 13 (APS4322-7000)/Term 14 (APS4322-5000)/FB Inputs/A{0..8 step 2} Y-Field <-> Data Pointer/HallSensorFieldsXYZ[{1..13 step 3}]  (5 links)
//     Term 13 (APS4322-7000)/Term 14 (APS4322-5000)/FB Inputs/A{0..8 step 2} Z-Field <-> Data Pointer/HallSensorFieldsXYZ[{2..14 step 3}]  (5 links)
//     Term 13 (APS4322-7000)/Term 14 (APS4322-5000)/FB Inputs/B{1..9 step 2} X-Field <-> Data Pointer/HallSensorFieldsXYZ[{15..27 step 3}]  (5 links)
//     Term 13 (APS4322-7000)/Term 14 (APS4322-5000)/FB Inputs/B{1..9 step 2} Y-Field <-> Data Pointer/HallSensorFieldsXYZ[{16..28 step 3}]  (5 links)
//     Term 13 (APS4322-7000)/Term 14 (APS4322-5000)/FB Inputs/B{1..9 step 2} Z-Field <-> Data Pointer/HallSensorFieldsXYZ[{17..29 step 3}]  (5 links)
//     Term 13 (APS4322-7000)/Term 14 (APS4322-5000)/FB Inputs/C{0..8 step 2} X-Field <-> Data Pointer/HallSensorFieldsXYZ[{30..42 step 3}]  (5 links)
//     Term 13 (APS4322-7000)/Term 14 (APS4322-5000)/FB Inputs/C{0..8 step 2} Y-Field <-> Data Pointer/HallSensorFieldsXYZ[{31..43 step 3}]  (5 links)
//     Term 13 (APS4322-7000)/Term 14 (APS4322-5000)/FB Inputs/C{0..8 step 2} Z-Field <-> Data Pointer/HallSensorFieldsXYZ[{32..44 step 3}]  (5 links)
//     Term 13 (APS4322-7000)/Term 14 (APS4322-5000)/FB Inputs/D{1..9 step 2} X-Field <-> Data Pointer/HallSensorFieldsXYZ[{45..57 step 3}]  (5 links)
//     Term 13 (APS4322-7000)/Term 14 (APS4322-5000)/FB Inputs/D{1..9 step 2} Y-Field <-> Data Pointer/HallSensorFieldsXYZ[{46..58 step 3}]  (5 links)
//     Term 13 (APS4322-7000)/Term 14 (APS4322-5000)/FB Inputs/D{1..9 step 2} Z-Field <-> Data Pointer/HallSensorFieldsXYZ[{47..59 step 3}]  (5 links)
//     Term 13 (APS4322-7000)/Term 14 (APS4322-5000)/FB Inputs/E{0..8 step 2} X-Field <-> Data Pointer/HallSensorFieldsXYZ[{60..72 step 3}]  (5 links)
//     Term 13 (APS4322-7000)/Term 14 (APS4322-5000)/FB Inputs/E{0..8 step 2} Y-Field <-> Data Pointer/HallSensorFieldsXYZ[{61..73 step 3}]  (5 links)
//     Term 13 (APS4322-7000)/Term 14 (APS4322-5000)/FB Inputs/E{0..8 step 2} Z-Field <-> Data Pointer/HallSensorFieldsXYZ[{62..74 step 3}]  (5 links)
//     Term 13 (APS4322-7000)/Term 14 (APS4322-5000)/FB Inputs/F{1..9 step 2} X-Field <-> Data Pointer/HallSensorFieldsXYZ[{75..87 step 3}]  (5 links)
//     Term 13 (APS4322-7000)/Term 14 (APS4322-5000)/FB Inputs/F{1..9 step 2} Y-Field <-> Data Pointer/HallSensorFieldsXYZ[{76..88 step 3}]  (5 links)
//     Term 13 (APS4322-7000)/Term 14 (APS4322-5000)/FB Inputs/F{1..9 step 2} Z-Field <-> Data Pointer/HallSensorFieldsXYZ[{77..89 step 3}]  (5 links)
//     Term 13 (APS4322-7000)/Term 14 (APS4322-5000)/FB Inputs/G{0..8 step 2} X-Field <-> Data Pointer/HallSensorFieldsXYZ[{90..102 step 3}]  (5 links)
//     Term 13 (APS4322-7000)/Term 14 (APS4322-5000)/FB Inputs/G{0..8 step 2} Y-Field <-> Data Pointer/HallSensorFieldsXYZ[{91..103 step 3}]  (5 links)
//     Term 13 (APS4322-7000)/Term 14 (APS4322-5000)/FB Inputs/G{0..8 step 2} Z-Field <-> Data Pointer/HallSensorFieldsXYZ[{92..104 step 3}]  (5 links)
//     Term 13 (APS4322-7000)/Term 14 (APS4322-5000)/FB Inputs/H{1..9 step 2} X-Field <-> Data Pointer/HallSensorFieldsXYZ[{105..117 step 3}]  (5 links)
//     Term 13 (APS4322-7000)/Term 14 (APS4322-5000)/FB Inputs/H{1..9 step 2} Y-Field <-> Data Pointer/HallSensorFieldsXYZ[{106..118 step 3}]  (5 links)
//     Term 13 (APS4322-7000)/Term 14 (APS4322-5000)/FB Inputs/H{1..9 step 2} Z-Field <-> Data Pointer/HallSensorFieldsXYZ[{107..119 step 3}]  (5 links)
//     Term 13 (APS4322-7000)/Term 14 (APS4322-5000)/FB Inputs/I{0..8 step 2} X-Field <-> Data Pointer/HallSensorFieldsXYZ[{120..132 step 3}]  (5 links)
//     Term 13 (APS4322-7000)/Term 14 (APS4322-5000)/FB Inputs/I{0..8 step 2} Y-Field <-> Data Pointer/HallSensorFieldsXYZ[{121..133 step 3}]  (5 links)
//     Term 13 (APS4322-7000)/Term 14 (APS4322-5000)/FB Inputs/I{0..8 step 2} Z-Field <-> Data Pointer/HallSensorFieldsXYZ[{122..134 step 3}]  (5 links)
//     Term 13 (APS4322-7000)/Term 14 (APS4322-5000)/FB Inputs/J{1..9 step 2} X-Field <-> Data Pointer/HallSensorFieldsXYZ[{135..147 step 3}]  (5 links)
//     Term 13 (APS4322-7000)/Term 14 (APS4322-5000)/FB Inputs/J{1..9 step 2} Y-Field <-> Data Pointer/HallSensorFieldsXYZ[{136..148 step 3}]  (5 links)
//     Term 13 (APS4322-7000)/Term 14 (APS4322-5000)/FB Inputs/J{1..9 step 2} Z-Field <-> Data Pointer/HallSensorFieldsXYZ[{137..149 step 3}]  (5 links)
//     Term 13 (APS4322-7000)/Term 14 (APS4322-5000)/FB Inputs/Status <-> Data Pointer/FeedbackStatus
//   Device 6 (EtherCAT) <-> TcCOM Objects/XPlanar/Part1/Tile12
//     Term 15 (APS4322-7000)/APS Comm Inputs/CommStatusWord <-> Data Pointer/MoverCommStatusWord
//     Term 15 (APS4322-7000)/APS Comm Inputs/Data {1..4} <-> Data Pointer/MoverCommDataIn[{0..3}]  (4 links)
//     Term 15 (APS4322-7000)/APS Comm Outputs/CommControlWord <-> Data Pointer/MoverCommControlWord
//     Term 15 (APS4322-7000)/APS Comm Outputs/Data 1 <-> Data Pointer/MoverCommDataOut
//     Term 15 (APS4322-7000)/APS Diagdata/DC Link Voltage <-> Data Pointer/DcLinkVoltage
//     Term 15 (APS4322-7000)/APS Diagdata/Power supply current <-> Data Pointer/PowerSupplyCurrent
//     Term 15 (APS4322-7000)/APS Inputs/StatusWord <-> Data Pointer/PowerUnitStatusWord
//     Term 15 (APS4322-7000)/APS Outputs/ControlWord <-> Data Pointer/PowerUnitControlWord
//     Term 15 (APS4322-7000)/APS Outputs/Current D 0X0 <-> Data Pointer/DCurrentSetPoints[0]
//     Term 15 (APS4322-7000)/APS Outputs/Current D 0X1 <-> Data Pointer/DCurrentSetPoints[1]
//     Term 15 (APS4322-7000)/APS Outputs/Current D 0X2 <-> Data Pointer/DCurrentSetPoints[2]
//     Term 15 (APS4322-7000)/APS Outputs/Current D 1X0 <-> Data Pointer/DCurrentSetPoints[6]
//     Term 15 (APS4322-7000)/APS Outputs/Current D 1X1 <-> Data Pointer/DCurrentSetPoints[7]
//     Term 15 (APS4322-7000)/APS Outputs/Current D 1X2 <-> Data Pointer/DCurrentSetPoints[8]
//     Term 15 (APS4322-7000)/APS Outputs/Current D 2X0 <-> Data Pointer/DCurrentSetPoints[12]
//     Term 15 (APS4322-7000)/APS Outputs/Current D 2X1 <-> Data Pointer/DCurrentSetPoints[13]
//     Term 15 (APS4322-7000)/APS Outputs/Current D 2X2 <-> Data Pointer/DCurrentSetPoints[14]
//     Term 15 (APS4322-7000)/APS Outputs/Current D 3X0 <-> Data Pointer/DCurrentSetPoints[18]
//     Term 15 (APS4322-7000)/APS Outputs/Current D 3X1 <-> Data Pointer/DCurrentSetPoints[19]
//     Term 15 (APS4322-7000)/APS Outputs/Current D 3X2 <-> Data Pointer/DCurrentSetPoints[20]
//     Term 15 (APS4322-7000)/APS Outputs/Current D 0Y0 <-> Data Pointer/DCurrentSetPoints[3]
//     Term 15 (APS4322-7000)/APS Outputs/Current D 0Y1 <-> Data Pointer/DCurrentSetPoints[4]
//     Term 15 (APS4322-7000)/APS Outputs/Current D 0Y2 <-> Data Pointer/DCurrentSetPoints[5]
//     Term 15 (APS4322-7000)/APS Outputs/Current D 1Y0 <-> Data Pointer/DCurrentSetPoints[9]
//     Term 15 (APS4322-7000)/APS Outputs/Current D 1Y1 <-> Data Pointer/DCurrentSetPoints[10]
//     Term 15 (APS4322-7000)/APS Outputs/Current D 1Y2 <-> Data Pointer/DCurrentSetPoints[11]
//     Term 15 (APS4322-7000)/APS Outputs/Current D 2Y0 <-> Data Pointer/DCurrentSetPoints[15]
//     Term 15 (APS4322-7000)/APS Outputs/Current D 2Y1 <-> Data Pointer/DCurrentSetPoints[16]
//     Term 15 (APS4322-7000)/APS Outputs/Current D 2Y2 <-> Data Pointer/DCurrentSetPoints[17]
//     Term 15 (APS4322-7000)/APS Outputs/Current D 3Y0 <-> Data Pointer/DCurrentSetPoints[21]
//     Term 15 (APS4322-7000)/APS Outputs/Current D 3Y1 <-> Data Pointer/DCurrentSetPoints[22]
//     Term 15 (APS4322-7000)/APS Outputs/Current D 3Y2 <-> Data Pointer/DCurrentSetPoints[23]
//     Term 15 (APS4322-7000)/APS Outputs/Current Q 0X0 <-> Data Pointer/QCurrentSetPoints[0]
//     Term 15 (APS4322-7000)/APS Outputs/Current Q 0X1 <-> Data Pointer/QCurrentSetPoints[1]
//     Term 15 (APS4322-7000)/APS Outputs/Current Q 0X2 <-> Data Pointer/QCurrentSetPoints[2]
//     Term 15 (APS4322-7000)/APS Outputs/Current Q 1X0 <-> Data Pointer/QCurrentSetPoints[6]
//     Term 15 (APS4322-7000)/APS Outputs/Current Q 1X1 <-> Data Pointer/QCurrentSetPoints[7]
//     Term 15 (APS4322-7000)/APS Outputs/Current Q 1X2 <-> Data Pointer/QCurrentSetPoints[8]
//     Term 15 (APS4322-7000)/APS Outputs/Current Q 2X0 <-> Data Pointer/QCurrentSetPoints[12]
//     Term 15 (APS4322-7000)/APS Outputs/Current Q 2X1 <-> Data Pointer/QCurrentSetPoints[13]
//     Term 15 (APS4322-7000)/APS Outputs/Current Q 2X2 <-> Data Pointer/QCurrentSetPoints[14]
//     Term 15 (APS4322-7000)/APS Outputs/Current Q 3X0 <-> Data Pointer/QCurrentSetPoints[18]
//     Term 15 (APS4322-7000)/APS Outputs/Current Q 3X1 <-> Data Pointer/QCurrentSetPoints[19]
//     Term 15 (APS4322-7000)/APS Outputs/Current Q 3X2 <-> Data Pointer/QCurrentSetPoints[20]
//     Term 15 (APS4322-7000)/APS Outputs/Current Q 0Y0 <-> Data Pointer/QCurrentSetPoints[3]
//     Term 15 (APS4322-7000)/APS Outputs/Current Q 0Y1 <-> Data Pointer/QCurrentSetPoints[4]
//     Term 15 (APS4322-7000)/APS Outputs/Current Q 0Y2 <-> Data Pointer/QCurrentSetPoints[5]
//     Term 15 (APS4322-7000)/APS Outputs/Current Q 1Y0 <-> Data Pointer/QCurrentSetPoints[9]
//     Term 15 (APS4322-7000)/APS Outputs/Current Q 1Y1 <-> Data Pointer/QCurrentSetPoints[10]
//     Term 15 (APS4322-7000)/APS Outputs/Current Q 1Y2 <-> Data Pointer/QCurrentSetPoints[11]
//     Term 15 (APS4322-7000)/APS Outputs/Current Q 2Y0 <-> Data Pointer/QCurrentSetPoints[15]
//     Term 15 (APS4322-7000)/APS Outputs/Current Q 2Y1 <-> Data Pointer/QCurrentSetPoints[16]
//     Term 15 (APS4322-7000)/APS Outputs/Current Q 2Y2 <-> Data Pointer/QCurrentSetPoints[17]
//     Term 15 (APS4322-7000)/APS Outputs/Current Q 3Y0 <-> Data Pointer/QCurrentSetPoints[21]
//     Term 15 (APS4322-7000)/APS Outputs/Current Q 3Y1 <-> Data Pointer/QCurrentSetPoints[22]
//     Term 15 (APS4322-7000)/APS Outputs/Current Q 3Y2 <-> Data Pointer/QCurrentSetPoints[23]
//     Term 15 (APS4322-7000)/APS Outputs/PhiE 0X0 <-> Data Pointer/PhiSetPoints[0]
//     Term 15 (APS4322-7000)/APS Outputs/PhiE 0X1 <-> Data Pointer/PhiSetPoints[1]
//     Term 15 (APS4322-7000)/APS Outputs/PhiE 0X2 <-> Data Pointer/PhiSetPoints[2]
//     Term 15 (APS4322-7000)/APS Outputs/PhiE 1X0 <-> Data Pointer/PhiSetPoints[6]
//     Term 15 (APS4322-7000)/APS Outputs/PhiE 1X1 <-> Data Pointer/PhiSetPoints[7]
//     Term 15 (APS4322-7000)/APS Outputs/PhiE 1X2 <-> Data Pointer/PhiSetPoints[8]
//     Term 15 (APS4322-7000)/APS Outputs/PhiE 2X0 <-> Data Pointer/PhiSetPoints[12]
//     Term 15 (APS4322-7000)/APS Outputs/PhiE 2X1 <-> Data Pointer/PhiSetPoints[13]
//     Term 15 (APS4322-7000)/APS Outputs/PhiE 2X2 <-> Data Pointer/PhiSetPoints[14]
//     Term 15 (APS4322-7000)/APS Outputs/PhiE 3X0 <-> Data Pointer/PhiSetPoints[18]
//     Term 15 (APS4322-7000)/APS Outputs/PhiE 3X1 <-> Data Pointer/PhiSetPoints[19]
//     Term 15 (APS4322-7000)/APS Outputs/PhiE 3X2 <-> Data Pointer/PhiSetPoints[20]
//     Term 15 (APS4322-7000)/APS Outputs/PhiE 0Y0 <-> Data Pointer/PhiSetPoints[3]
//     Term 15 (APS4322-7000)/APS Outputs/PhiE 0Y1 <-> Data Pointer/PhiSetPoints[4]
//     Term 15 (APS4322-7000)/APS Outputs/PhiE 0Y2 <-> Data Pointer/PhiSetPoints[5]
//     Term 15 (APS4322-7000)/APS Outputs/PhiE 1Y0 <-> Data Pointer/PhiSetPoints[9]
//     Term 15 (APS4322-7000)/APS Outputs/PhiE 1Y1 <-> Data Pointer/PhiSetPoints[10]
//     Term 15 (APS4322-7000)/APS Outputs/PhiE 1Y2 <-> Data Pointer/PhiSetPoints[11]
//     Term 15 (APS4322-7000)/APS Outputs/PhiE 2Y0 <-> Data Pointer/PhiSetPoints[15]
//     Term 15 (APS4322-7000)/APS Outputs/PhiE 2Y1 <-> Data Pointer/PhiSetPoints[16]
//     Term 15 (APS4322-7000)/APS Outputs/PhiE 2Y2 <-> Data Pointer/PhiSetPoints[17]
//     Term 15 (APS4322-7000)/APS Outputs/PhiE 3Y0 <-> Data Pointer/PhiSetPoints[21]
//     Term 15 (APS4322-7000)/APS Outputs/PhiE 3Y1 <-> Data Pointer/PhiSetPoints[22]
//     Term 15 (APS4322-7000)/APS Outputs/PhiE 3Y2 <-> Data Pointer/PhiSetPoints[23]
//     Term 15 (APS4322-7000)/Term 16 (APS4322-5000)/FB Inputs/A{0..8 step 2} X-Field <-> Data Pointer/HallSensorFieldsXYZ[{0..12 step 3}]  (5 links)
//     Term 15 (APS4322-7000)/Term 16 (APS4322-5000)/FB Inputs/A{0..8 step 2} Y-Field <-> Data Pointer/HallSensorFieldsXYZ[{1..13 step 3}]  (5 links)
//     Term 15 (APS4322-7000)/Term 16 (APS4322-5000)/FB Inputs/A{0..8 step 2} Z-Field <-> Data Pointer/HallSensorFieldsXYZ[{2..14 step 3}]  (5 links)
//     Term 15 (APS4322-7000)/Term 16 (APS4322-5000)/FB Inputs/B{1..9 step 2} X-Field <-> Data Pointer/HallSensorFieldsXYZ[{15..27 step 3}]  (5 links)
//     Term 15 (APS4322-7000)/Term 16 (APS4322-5000)/FB Inputs/B{1..9 step 2} Y-Field <-> Data Pointer/HallSensorFieldsXYZ[{16..28 step 3}]  (5 links)
//     Term 15 (APS4322-7000)/Term 16 (APS4322-5000)/FB Inputs/B{1..9 step 2} Z-Field <-> Data Pointer/HallSensorFieldsXYZ[{17..29 step 3}]  (5 links)
//     Term 15 (APS4322-7000)/Term 16 (APS4322-5000)/FB Inputs/C{0..8 step 2} X-Field <-> Data Pointer/HallSensorFieldsXYZ[{30..42 step 3}]  (5 links)
//     Term 15 (APS4322-7000)/Term 16 (APS4322-5000)/FB Inputs/C{0..8 step 2} Y-Field <-> Data Pointer/HallSensorFieldsXYZ[{31..43 step 3}]  (5 links)
//     Term 15 (APS4322-7000)/Term 16 (APS4322-5000)/FB Inputs/C{0..8 step 2} Z-Field <-> Data Pointer/HallSensorFieldsXYZ[{32..44 step 3}]  (5 links)
//     Term 15 (APS4322-7000)/Term 16 (APS4322-5000)/FB Inputs/D{1..9 step 2} X-Field <-> Data Pointer/HallSensorFieldsXYZ[{45..57 step 3}]  (5 links)
//     Term 15 (APS4322-7000)/Term 16 (APS4322-5000)/FB Inputs/D{1..9 step 2} Y-Field <-> Data Pointer/HallSensorFieldsXYZ[{46..58 step 3}]  (5 links)
//     Term 15 (APS4322-7000)/Term 16 (APS4322-5000)/FB Inputs/D{1..9 step 2} Z-Field <-> Data Pointer/HallSensorFieldsXYZ[{47..59 step 3}]  (5 links)
//     Term 15 (APS4322-7000)/Term 16 (APS4322-5000)/FB Inputs/E{0..8 step 2} X-Field <-> Data Pointer/HallSensorFieldsXYZ[{60..72 step 3}]  (5 links)
//     Term 15 (APS4322-7000)/Term 16 (APS4322-5000)/FB Inputs/E{0..8 step 2} Y-Field <-> Data Pointer/HallSensorFieldsXYZ[{61..73 step 3}]  (5 links)
//     Term 15 (APS4322-7000)/Term 16 (APS4322-5000)/FB Inputs/E{0..8 step 2} Z-Field <-> Data Pointer/HallSensorFieldsXYZ[{62..74 step 3}]  (5 links)
//     Term 15 (APS4322-7000)/Term 16 (APS4322-5000)/FB Inputs/F{1..9 step 2} X-Field <-> Data Pointer/HallSensorFieldsXYZ[{75..87 step 3}]  (5 links)
//     Term 15 (APS4322-7000)/Term 16 (APS4322-5000)/FB Inputs/F{1..9 step 2} Y-Field <-> Data Pointer/HallSensorFieldsXYZ[{76..88 step 3}]  (5 links)
//     Term 15 (APS4322-7000)/Term 16 (APS4322-5000)/FB Inputs/F{1..9 step 2} Z-Field <-> Data Pointer/HallSensorFieldsXYZ[{77..89 step 3}]  (5 links)
//     Term 15 (APS4322-7000)/Term 16 (APS4322-5000)/FB Inputs/G{0..8 step 2} X-Field <-> Data Pointer/HallSensorFieldsXYZ[{90..102 step 3}]  (5 links)
//     Term 15 (APS4322-7000)/Term 16 (APS4322-5000)/FB Inputs/G{0..8 step 2} Y-Field <-> Data Pointer/HallSensorFieldsXYZ[{91..103 step 3}]  (5 links)
//     Term 15 (APS4322-7000)/Term 16 (APS4322-5000)/FB Inputs/G{0..8 step 2} Z-Field <-> Data Pointer/HallSensorFieldsXYZ[{92..104 step 3}]  (5 links)
//     Term 15 (APS4322-7000)/Term 16 (APS4322-5000)/FB Inputs/H{1..9 step 2} X-Field <-> Data Pointer/HallSensorFieldsXYZ[{105..117 step 3}]  (5 links)
//     Term 15 (APS4322-7000)/Term 16 (APS4322-5000)/FB Inputs/H{1..9 step 2} Y-Field <-> Data Pointer/HallSensorFieldsXYZ[{106..118 step 3}]  (5 links)
//     Term 15 (APS4322-7000)/Term 16 (APS4322-5000)/FB Inputs/H{1..9 step 2} Z-Field <-> Data Pointer/HallSensorFieldsXYZ[{107..119 step 3}]  (5 links)
//     Term 15 (APS4322-7000)/Term 16 (APS4322-5000)/FB Inputs/I{0..8 step 2} X-Field <-> Data Pointer/HallSensorFieldsXYZ[{120..132 step 3}]  (5 links)
//     Term 15 (APS4322-7000)/Term 16 (APS4322-5000)/FB Inputs/I{0..8 step 2} Y-Field <-> Data Pointer/HallSensorFieldsXYZ[{121..133 step 3}]  (5 links)
//     Term 15 (APS4322-7000)/Term 16 (APS4322-5000)/FB Inputs/I{0..8 step 2} Z-Field <-> Data Pointer/HallSensorFieldsXYZ[{122..134 step 3}]  (5 links)
//     Term 15 (APS4322-7000)/Term 16 (APS4322-5000)/FB Inputs/J{1..9 step 2} X-Field <-> Data Pointer/HallSensorFieldsXYZ[{135..147 step 3}]  (5 links)
//     Term 15 (APS4322-7000)/Term 16 (APS4322-5000)/FB Inputs/J{1..9 step 2} Y-Field <-> Data Pointer/HallSensorFieldsXYZ[{136..148 step 3}]  (5 links)
//     Term 15 (APS4322-7000)/Term 16 (APS4322-5000)/FB Inputs/J{1..9 step 2} Z-Field <-> Data Pointer/HallSensorFieldsXYZ[{137..149 step 3}]  (5 links)
//     Term 15 (APS4322-7000)/Term 16 (APS4322-5000)/FB Inputs/Status <-> Data Pointer/FeedbackStatus
//   Device 6 (EtherCAT) <-> TcCOM Objects/XPlanar/Part1/Tile3
//     Term 5 (APS4322-7000)/APS Comm Inputs/CommStatusWord <-> Data Pointer/MoverCommStatusWord
//     Term 5 (APS4322-7000)/APS Comm Inputs/Data {1..4} <-> Data Pointer/MoverCommDataIn[{0..3}]  (4 links)
//     Term 5 (APS4322-7000)/APS Comm Outputs/CommControlWord <-> Data Pointer/MoverCommControlWord
//     Term 5 (APS4322-7000)/APS Comm Outputs/Data 1 <-> Data Pointer/MoverCommDataOut
//     Term 5 (APS4322-7000)/APS Diagdata/DC Link Voltage <-> Data Pointer/DcLinkVoltage
//     Term 5 (APS4322-7000)/APS Diagdata/Power supply current <-> Data Pointer/PowerSupplyCurrent
//     Term 5 (APS4322-7000)/APS Inputs/StatusWord <-> Data Pointer/PowerUnitStatusWord
//     Term 5 (APS4322-7000)/APS Outputs/ControlWord <-> Data Pointer/PowerUnitControlWord
//     Term 5 (APS4322-7000)/APS Outputs/Current D 0X0 <-> Data Pointer/DCurrentSetPoints[0]
